// TIA Portal project "MAGNET_ITLK_V15.1" (V15.1)
// Interlocs logic fot the CERN magnet tests

(* hardware
DEVICE "S71500/ET200MP station_1"  S7-1500 station
   slot 0: "Rail_0"  Rack  6ES7 590-1***0-0AA0
   slot 0: "PS 25W 24VDC_1"  PS 25W 24VDC  6ES7 505-0KA00-0AB0  V1.0
   slot 1: "PLC_1"  CPU 1511F-1 PN  6ES7 511-1FK02-0AB0  V2.6
      slot 3: "CPU display_1"  6ES7591-1AA00-0AA0
   slot 2: "DI 32x24VDC HF_1"  DI 32x24VDC HF  6ES7 521-1BL00-0AB0  V2.0
   slot 3: "DQ 32x24VDC/0.5A HF_1"  DQ 32x24VDC/0.5A HF  6ES7 522-1BL01-0AB0  V1.1
   slot 100: "PM 70W 120/230VAC"  PM 70W 120/230VAC  6EP1332-4BA00
*)

// ===== PLC "PLC_1"  CPU 1511F-1 PN =====

VAR_GLOBAL   // PLC tag table "Default tag table"
   "Clock_Byte" AT %MB0 : Byte;
   "Clock_10Hz" AT %M0.0 : Bool;
   "Clock_5Hz" AT %M0.1 : Bool;
   "Clock_2.5Hz" AT %M0.2 : Bool;
   "Clock_2Hz" AT %M0.3 : Bool;
   "Clock_1.25Hz" AT %M0.4 : Bool;
   "Clock_1Hz" AT %M0.5 : Bool;
   "Clock_0.625Hz" AT %M0.6 : Bool;
   "Clock_0.5Hz" AT %M0.7 : Bool;
END_VAR

VAR_GLOBAL CONSTANT   // PLC tag table "ConstDiagnostics"
   "DEV_STATE_OK" : USInt := 1;   // device state ok
   "DEV_STATE_LOST_CON" : USInt := 3;   // device state lost connection
   "DEV_STATE_DISABLED" : USInt := 4;   // device state device disabled
   "DEV_STATE_WAS_FAULT" : USInt := 12;   // device state was fault
   "DEV_STATE_WAS_LOST" : USInt := 13;   // device state connection was lost
   "DEV_STATE_WAS_DISABLED" : USInt := 14;   // device state device was disabled
   "MAX_DEVICES_SYSTEM" : Int := 10;   // max number of devices per IO system
   "MAX_MODULES_DEVICE" : Int := 20;   // max number of modules per device
   "MAX_MODULES_LOCAL" : Int := 15;   // max number of local modules
   "LAST_DEVICE" : Int := -1;   // no next device
   "MAX_SYSTEM" : Int := 2;   // max number of IO system in the project / max number of devices per IO system
   "IO_SYSTEM1" : Int := 1;   // index for IO system 1
   "IO_SYSTEM2" : Int := 2;   // index for IO system 2
   "IO_SYSTEM0" : Int := 0;   // index for local PLC
   "DEV_STATE_FAULT" : USInt := 2;   // device state fault
END_VAR

VAR_GLOBAL   // PLC tag table "ai_dio_tag"
   "DC24V_AUX1_OK" AT %I3.5 : Bool;
   "FLSHBX_HE" AT %Q1.3 : Bool;   // Flashbox Helium
   "KLY_IP_ISn_Current_01" AT %IW304 : Int;
   "KLY_IP_ISn_Current_02" AT %IW306 : Int;
   "KLY_Oil_TSn_SurfTemp" AT %IW222 : Int;
   "KLY_Oil_FSn_WatOutletFlow" AT %IW238 : Int;
   "KLY_Sol_TSn_WatInletTemp" AT %IW216 : Int;
   "KLY_Sol_TSn_WatOutletTemp" AT %IW218 : Int;
   "KLY_Sol_FSn_WatOutletFlow" AT %IW236 : Int;
   "KLY_Sol_TSn_SurfTemp" AT %IW220 : Int;
   "KLY_Win_FSn_WatOutletFlow" AT %IW254 : Int;
   "KLY_Win_TSn_WatOutletTemp" AT %IW214 : Int;
   "KLY_Win_TSn_WatOutletSleeveTemp" AT %IW212 : Int;
   "KLY_Coll_TSn_TopTemp" AT %IW224 : Int;
   "KLY_Coll_TSn_EdgeTemp" AT %IW226 : Int;
   "KLY_Coll_TSn_WatInletTemp" AT %IW248 : Int;
   "KLY_Coll_TSn_WatOutletTemp" AT %IW252 : Int;
   "KLY_Coll_FSn_WatOutletFlow" AT %IW232 : Int;
   "KLY_Body_TSn_WatInletTemp" AT %IW204 : Int;
   "KLY_Body_TSn_WatOutletTemp" AT %IW206 : Int;
   "KLY_Body_FSn_WatOutletFlow" AT %IW234 : Int;
   "KLY_Coll_CollDissipation" AT %IW240 : Int;
   "KLY_Body_BodyDisssipation" AT %IW242 : Int;
   "RFDS_Load_FSn_WatOutletFlow" AT %IW256 : Int;
   "RFDS_Load_TSn_WatOutletTemp" AT %IW250 : Int;
   "spare(7)" AT %Q3.3 : Bool;
   "NO_QUENCH" AT %I3.7 : Bool;   // No quench detected (from safety matrix)
   "DAQ_OK" AT %I1.7 : Bool;   // DAQ system OK
   "PC_1_POWER_FAILURE" AT %I0.6 : Bool;   // Power converter status
   "EE_1_PC_SPA_OK" AT %I0.5 : Bool;   // Slow Power Abort switch OK
   "EE_1_REMOTE" AT %I0.1 : Bool;   // Energy extractionswitches are in remote
   "EE_1_NO_ERROR_CL" AT %I0.2 : Bool;   // Energy extraction switches have nointernalerrors
   "EE_1_CLOSED" AT %I0.3 : Bool;   // Energy extraction keys are closed
   "EE_1_POWER_PERM" AT %I0.0 : Bool;   // Energy extraction switches give power permit
   "KEY2_OK" AT %I1.6 : Bool;   // Cable in parking (0)/ operation (1) position
   "PC_1_CONNECT" AT %I0.7 : Bool;   // Power converter connected (closed contact)
   "PC_1_EXT_OUT" AT %I1.0 : Bool;   // Status of the main circuit breaker of the pwr converter
   "KEY1_OK" AT %I1.5 : Bool;   // Emergency Button OK
   "EE_1_NO_WARNING" AT %I0.4 : Bool;   // Energy Extraction not in warning condition
   "EE_1_FS" AT %I1.1 : Bool;   // EE_1 water flow switch
   "POLSW_1_POS1" AT %I1.2 : Bool;   // Polarity switch 1 position 1
   "EE_2_FS" AT %I3.1 : Bool;   // EE _1water flow switch
   "POLSW_2_POS1" AT %I3.2 : Bool;   // Polarity switch position 1
   "DC24V_AUX2_OK" AT %I3.6 : Bool;   // 24 V PLC power supply ok
   "POLSW_2_POS2" AT %I3.3 : Bool;   // Polarity switch position 2
   "spare(2_4)" AT %I3.4 : Bool;
   "spare3" AT %Q1.0 : Bool;   // Direct power abort
   "PC_1_PERMIT" AT %Q0.3 : Bool;   // Powerconverter permit
   "PC_1_EXT" AT %Q0.4 : Bool;   // Fast Power Abort
   "CLOSE_EE_1" AT %Q0.1 : Bool;   // Close energy extraction switch (action by the operator)
   "EE_1_OPEN_RQ" AT %Q0.0 : Bool;   // Request to open energy extraction switch
   "RESET_EE_1" AT %Q0.2 : Bool;   // Reset energy extraction switch (action by the operator)
   "FLSHBX_HVOLT" AT %Q1.1 : Bool;   // Flashbox High Voltage
   "FLSHBX_HCUR" AT %Q1.2 : Bool;   // Flashbox High Current
   "CPU_Send_RQ" AT %Q3.7 : Bool;
   "MemByteClock7" AT %Q3.6 : Bool;
   "EE_2_OPEN_RQ" AT %Q2.0 : Bool;   // Request to open energy extraction switch
   "CLOSE_EE_2" AT %Q2.1 : Bool;   // Close energy extraction switch (action by the operator)
   "RESET_EE_2" AT %Q2.2 : Bool;   // Reset energy extraction switch (action by the operator)
   "PC_2_PERMIT" AT %Q2.3 : Bool;   // Powerconverter permit
   "PC_2_EXT" AT %Q2.4 : Bool;   // Fast Power Abort
   "EE_2_POWER_PERM" AT %I2.0 : Bool;   // Energy extraction switches give power permit
   "EE_2_REMOTE" AT %I2.1 : Bool;   // Energy extractionswitches are in remote
   "EE_2_NO_ERROR_CL" AT %I2.2 : Bool;   // Energy extraction switches have nointernalerrors
   "EE_2_CLOSED" AT %I2.3 : Bool;   // Energy extraction keys are closed
   "EE_2_NO_WARNING" AT %I2.4 : Bool;   // Energy Extraction not in warning condition
   "EE_2_PC_SPA_OK" AT %I2.5 : Bool;   // Slow Power Abort switch OK
   "PC_2_POWER_FAILURE" AT %I2.6 : Bool;   // Power converter status
   "PC_2_CONNECT" AT %I2.7 : Bool;   // Power converter connected (closed contact)
   "PC_2_EXT_OUT" AT %I3.0 : Bool;   // Status of the main circuit breaker of the pwr converter
   "POLSW_1_POS2" AT %I1.3 : Bool;   // Polarity switch 1 position 2
   "spare(1_4)" AT %I1.4 : Bool;
END_VAR

VAR_GLOBAL CONSTANT   // PLC tag table "ai_dio_tag"
   "DI" : Byte := 1;   // Digital Input type
   "DO" : Byte := 2;   // Digital Output type
   "TSn" : Byte := 1;   // Temperature sensor type
   "PSn" : Byte := 2;   // Pressure sensor type
   "VSn_bipolar_50mV" : Byte := 20;
   "TSn_TC" : Byte := 11;   // Thermocouple - temperature sensor
   "VSn_bipolar_500mV" : Byte := 21;
   "VSn_bipolar_1V" : Byte := 22;
   "VSn_bipolar_5V" : Byte := 23;
   "VSn_bipolar_10V" : Byte := 24;
   "VSn_1_5v" : Byte := 25;
   "VSn_0_10v" : Byte := 3;   // Voltage sensor type
   "ISn_0_20mA" : Byte := 4;
   "ISn_4_20mA" : Byte := 5;
   "FSn_05_80_l_min" : Byte := 6;   // DU06.E.V.R015.A.0 Ultrasonic flowmeter
   "FSn_8_1000_l_min" : Byte := 7;   // DU06.E.V.R050.A.0 Ultrasonic flowmeter
   "PSn_0_10_bar" : Byte := 8;   // PMD02.E.15G.A75.S.I4.K2.0.0 Pressure sensor
   "TSn_0_50_C" : Byte := 9;   // TD20.117 14.111787 - Temperature sensor
   "ISn_bipolar_20mA" : Byte := 26;
   "TSn_PT100" : Byte := 10;   // PT100 - temperature sensor
   "UNKNOW" : Byte := 0;
   "COLL_DISP" : Byte := 12;   // Collector dissipation
   "BODY_DISP" : Byte := 13;   // Body dissipation
   "ISn_IP" : Byte := 27;
   "NORMAL_OPERATION" : Byte := 3;
   "NO_CONVERSION" : Byte := 255;   // Real type - do notdoany conversion
END_VAR

VAR_GLOBAL   // PLC tag table "IOs"
   "FIL_I_REG" AT %M300.0 : Bool;
   "FIL_VMON" AT %MW302 : Int;
   "FIL_IMON" AT %IW314 : Int;
   "FIL_WMON" AT %IW312 : Int;
   "FIL_OUT_LOC_REM" AT %M350.2 : Bool;
   "FIL_OUT_VPGM" AT %MW352 : Int;
   "FIL_START_COMMAND" AT %M300.4 : Bool;
   "FIL_STOP_COMMAND" AT %M300.5 : Bool;
   "SOL1_I_REG" AT %M308.0 : Bool;
   "SOL1_LOC_REM" AT %M308.2 : Bool;
   "SOL1_FAULT" AT %M308.3 : Bool;
   "SOL1_START_COMMAND" AT %M308.4 : Bool;
   "SOL1_STOP_COMMAND" AT %M308.5 : Bool;
   "SOL1_VMON" AT %IW296 : Int;
   "SOL1_IMON" AT %IW300 : Int;
   "SOL1_WMON" AT %MW304 : Int;
   "SOL1_OUT_RESET" AT %M356.1 : Bool;
   "SOL1_OUT_VPGM" AT %MW358 : Int;
   "SOL1_OUT_IPGM" AT %QW6 : Int;
   "FIL_OUT_IPGM" AT %QW4 : Int;
   "SOL2_OUT_IPGM" AT %QW8 : Int;
   "SOL2_VMON" AT %IW298 : Int;
   "SOL2_IMON" AT %IW302 : Int;
   "SOL2_START_COMMAND" AT %M308.6 : Bool;
   "SOL2_STOP_COMMAND" AT %M308.7 : Bool;
END_VAR

VAR_GLOBAL CONSTANT   // PLC tag table "IOs"
   "ENG_0-30A" : Byte := 30;
   "ENG_0-900W" : Byte := 31;
   "PSU_KLYSTRON_SOLENOID" : Int := 2;
   "ENG_0-17A" : Byte := 18;
   "ENG_0-300V" : Byte := 19;
END_VAR

VAR_GLOBAL   // PLC tag table "MachineState"
   "mbi_auxPre" AT %M7.0 : Bool;
   "mbi_filPre" AT %M7.1 : Bool;
   "mbi_stbyPre" AT %M7.3 : Bool;
   "mbi_hvonPre" AT %M7.4 : Bool;
   "mbi_rfonPre" AT %M7.5 : Bool;
   "mw_setState" AT %MW10 : Int;
   "mbi_auxSup" AT %M7.6 : Bool;
   "mbi_filSup" AT %M7.7 : Bool;
   "mbi_stbySup" AT %M8.0 : Bool;
   "mbi_hvonSup" AT %M8.1 : Bool;
   "mbi_rfonSup" AT %M8.2 : Bool;
   "mbi_filPreReady" AT %M7.2 : Bool;
   "mb_location" AT %MB20 : Byte;
   "mb_actState" AT %MB21 : Byte;
   "mbi_aux" AT %M8.4 : Bool;
   "mbi_fil" AT %M8.5 : Bool;
   "mbi_stdby" AT %M8.6 : Bool;
   "mbi_hvon" AT %M8.7 : Bool;
   "mbi_rfon" AT %M9.0 : Bool;
   "t_filHeatingDelay" AT %M9.1 : Bool;
   "t_auxSup" AT %T10 : Timer;
   "t_filSup" AT %T11 : Timer;
   "t_stdbySup" AT %T12 : Timer;
   "t_hvonSup" AT %T13 : Timer;
   "t_rfonSup" AT %T14 : Timer;
END_VAR

TYPE "CommParam"
VERSION : 0.1
   STRUCT
      interface_id : Word;   // HW-identifier of IE-interface submodule
      conn_id : Word;   // Connection reference / identifier
      connection_type : Byte := 16#000B;   // Type of connection: 11=TCP/IP, 19=UDP (17=TCP/IP) ??B#16#11??
      active_established : Bool := False;   // active/passive connection establishment
      local_port : UInt;   // local UDP/TCP port number
      init_com : Bool;   // send_db : INT; recv_db : INT;
      send_len : UDInt;
      recv_len : UDInt;
      sendtrigger : Bool;
      sendtime : Time;
      sendinterval : DInt;
   END_STRUCT;
END_TYPE

TYPE "PSU_Inputs"
VERSION : 0.1
   STRUCT
      I_REG : Bool;   // Signal from PSU, PSU is in constant current mode
      ON_STATUS : Bool;   // Signal from PSU, PSU is truned ON
      LOC_REM : Bool;   // Signal from PSU, TRUE=REMOTE,FALSE=LOCAL
      FAULT : Bool;   // Signal from PSU, TRUE=PSU OK
      VMON : Int;   // Value from PSU, Actual Voltage (V)
      IMON : Int;   // Value from PSU, Actual Current (I)
      WMON : Int;   // Value from PSU, Actual Power (W)
   END_STRUCT;
END_TYPE

TYPE "PSU_Outputs"
VERSION : 0.1
   STRUCT
      ENA_IN : Bool;   // Enable/Disable Power Supply
      RESET : Bool;   // Fault reset
      LOC_REM : Bool;   // LOCAL/REMOTE mode
      VPGM : Int;   // Voltage Setpoint
      IPGM : Int;   // Current Setpoint
   END_STRUCT;
END_TYPE

TYPE "FILAMENT_RST"
VERSION : 0.1
   STRUCT
      ON_STATUS : Bool;   // PSU is Operating normally
      STARTED : Bool;   // PSU has received the ON Command
      STOPPED : Bool;   // PSU is NOT operating
      WARMUP : Bool;   // PSU start procedure is running
      TEMP_REACHED : Bool;   // PSU is at operating temperature - Warmup Done
      I_REG : Bool;   // HIGH= the PSU is in constant cuttent mode
      LOC_REM_ST : Bool;   // HIGH=REMOTE,FALSE=LOCAL
      N_LATCH : Bool;   // Disable Latching from PLC code
      N_FORCE : Bool;   // Disable forcing from PLC code
      IsFIRST : Bool;   // Is the PSU Interlock the first Interlock?
      WARNING : Bool;   // PSU Warning Bit
      INTERLOCK : Bool;   // PSU Interlock Bit
      FORCE_ON : Bool;   // Feedback ForceON
      S_ON_STATUS : Bool;   // Feedback ON_STATUS input
      S_I_REG : Bool;   // Feedback I_REG input
      S_FAULT : Bool;   // Feedback FAULT input
      S_LOC_REM : Bool;   // Feedback LOC_REM input
      I_RAMP_ON : Bool;   // Feedback for Current Ramp ON
      V_RAMP_ON : Bool;   // Feedback for Voltage Ramp ON
      DTYP : Byte;   // PSU Type
      ERR : Word;   // Different error bits stored in the word descibed in the code
      TOTAL_WARMUP_LEFT : Real;   // How much time is left before operation
      WARMUP_LEFT_SP : Real;   // How much time is left before actual SetPoint reached
      UPTIME_NO_HV : Real;   // PSU uptime without HighVoltage
      TIME_COLD_SP1 : Real;   // Feedback Setpoint1 Time
      TIME_COLD_SP2 : Real;   // Feedback Setpoint2 Time
      TIME_COLD_SP3 : Real;   // Feedback Setpoint3 Time
      TIME_WARM_SP1 : Real;   // Feedback Setpoint1 Time warm
      TIME_WARM_SP2 : Real;   // Feedback Setpoint2 Time warm
      TIME_WARM_SP3 : Real;   // Feedback Setpoint3 Time warm
      ACT_SP : Real;   // Actual Setpoint number
      I_RAMP_RATE : Real;   // Feedback Calculated Current Ramp Rate
      V_RAMP_RATE : Real;   // Feedback Calculated Voltage Ramp Rate
      VMON : Real;   // Actual Voltage (V)
      IMON : Real;   // Actual Current (I)
      WMON : Real;   // Actual Power (W)
      S_VMON : Real;   // Feedback VMON input
      S_IMON : Real;   // Feedback IMON input
      S_WMON : Real;   // Feedback WMON input
      I_SP1 : Real;   // Feedback Setpoint1 Current
      I_SP2 : Real;   // Feedback Setpoint2 Current
      I_SP3 : Real;   // Feedback Setpoint3 Current
      V_SP1 : Real;   // Feedback Setpoint1 Voltage
      V_SP2 : Real;   // Feedback Setpoint2 Voltage
      V_SP3 : Real;   // Feedback Setpoint3 Voltage
      I_HIHI : Real;   // Feedback Current Alarm High
      I_LOLO : Real;   // Feedback Current Alarm Low
      I_HIGH : Real;   // Feedback Current Warning High
      I_LOW : Real;   // Feedback Current Warning Low
      W_HIHI : Real;   // Feedback Power Alarm High
      W_LOLO : Real;   // Feedback Power Alarm Low
      W_HIGH : Real;   // Feedback Power Warning High
      W_LOW : Real;   // Feedback Power Warning Low
      I_EGU_SP : Real;   // CurrentSetpoint in engunit
      FIL_MAX_I : Real;   // The maximum allowed Filament current hardwired in the PSU code
      FIL_MAX_W : Real;   // The maximum allowed Filament power hardwired in the PSU code
      TOL_InWARMUP : Real;   // Feedback for Tolareance during Warmup between IMON and IPGM
      TMPST : Date_And_Time;   // Last Interlock or Warning Timestamp
      TOTAL_WARMPUP_T : S5Time;   // Sum of the SetPoints time
   END_STRUCT;
END_TYPE

TYPE "CPU_WCONF"
VERSION : 0.0
   STRUCT
      RESET : Bool;   // CPU reset command
      OFF : Bool;   // OFF Command
      EE_1_CLOSE : Bool;   // Auxiliary Command
      EE_1_RESET : Bool;   // Filament Command
      EE_2_CLOSE : Bool;   // Standby command
      EE_2_RESET : Bool;   // High-voltage ON command
      RFON : Bool;   // RF ON command
      TEST_ALL_AD : Bool;   // Test all arc detectors
      WR_DATA : Bool;   // Write data into the read DB
      OP_MODE : Byte;   // 1 = Bypass mode, 2 = Maintenance/testing mode, 3 = Normal operation, 4 = Wire test
   END_STRUCT;
END_TYPE

TYPE "FILAMENT_WST"
VERSION : 0.1
   STRUCT
      START : Bool;   // Start PSU operation. TRUE=ENABLED
      STOP : Bool := false;   // Stop PSU and reset Timers TRUE = STOP
      FORCE : Bool;   // Force PSU block TRUE = FORCE all inputs
      S_ON_STATUS : Bool;   // Force ON_STATUS input
      S_IVAL : Bool;   // Force I_REG input
      S_LOC_REM : Bool;   // Force LOC_REM input
      S_FAULT : Bool;   // Force FAULT input
      I_RAMP_ON : Bool;   // Enable ramping for Current SP
      V_RAMP_ON : Bool;   // Enable ramping for Voltage SP
      RESET : Bool;   // Reset PSU
      WR_DATA : Bool;   // Write data into the read DB
      TIME_COLD_SP1 : Real;   // Setpoint1 Time
      TIME_COLD_SP2 : Real;   // Setpoint2 Time
      TIME_COLD_SP3 : Real;   // Setpoint3 Time
      TIME_WARM_SP1 : Real;   // Setpoint1 Time if the PSU is already warm
      TIME_WARM_SP2 : Real;   // Setpoint2 Time if the PSU is already warm
      TIME_WARM_SP3 : Real;   // Setpoint3 Time if the PSU is already warm
      I_SP1 : Real;   // Setpoint1 Current
      I_SP2 : Real;   // Setpoint2 Current
      I_SP3 : Real;   // Setpoint3 Current
      V_SP1 : Real;   // Setpoint1 Voltage
      V_SP2 : Real;   // Setpoint2 Voltage
      V_SP3 : Real;   // Setpoint3 Voltage
      S_VMON : Real;   // Force VMON input
      S_IMON : Real;   // Force IMON input
      S_WMON : Real;   // Force WMON input
      V_RAMP_RATE : Real;   // Voltage Ramp rate unit/sec (not used now)
      I_RAMP_RATE : Real;   // Current Ramp rate unit/sec (not used now)
      I_HIHI : Real;   // Current Alarm High
      I_LOLO : Real;   // Current Alarm Low
      I_HIGH : Real;   // Current Warning High
      I_LOW : Real;   // Current Warning Low
      W_HIHI : Real;   // Power Alarm High
      W_LOLO : Real;   // Power Alarm Low
      W_HIGH : Real;   // Power Warning High
      W_LOW : Real;   // Power Warning Low
      TOL_InWARMUP_SP : Real;   // Maximum allowed difference between IMON and IPGM
   END_STRUCT;
END_TYPE

TYPE "CPU_RCONF"
VERSION : 0.0
   STRUCT
      RESET : Bool;   // CPU reset command
      LATCH_MODE : Bool;   // CPU latching mode
      INTERLOCK : Bool;   // CPU Interlock/Alarm
      ACK_REQ : Bool;   // CPU Warning
      GERSEMI_COM_OK : Bool;   // Communication with Gersemi OK
      FLSHBX_HV : Bool;   // Flash Box High Voltage
      FLSHBX_HC : Bool;   // Flash Box High Current
      FLSHBX_He : Bool;   // Flash Box Helium
      RFON_MISS_COND : Bool;   // RF Enable missed condition
      AUX_SUP_COND : Bool;   // AUX missed supervision
      FIL_SUP_COND : Bool;   // FIL missed supervision
      STDBY_SUP_COND : Bool;   // STDBY missed supervision
      HVON_SUP_COND : Bool;   // HVON missed supervision
      RFON_SUP_COND : Bool;   // RFON missed supervision
      OFF : Bool;   // OFF Command
      EE_1_CLOSE : Bool;   // Auxiliary Command
      EE_1_RESET : Bool;   // Filament Command
      EE_2_CLOSE : Bool;   // Standby command
      EE_2_RESET : Bool;   // High-voltage ON command
      RFON : Bool;   // RF ON command
      FORCE_DIS_MODE_ACT : Bool;   // One or more signals are being disabled or forced
      TEST_ALL_AD : Bool;   // Test all arc detectors
      ACT_STAT : Byte;   // Actual State
      SET_STATE : Int;   // Set State to the target
      OP_MODE : Byte;   // 1 = Bypass mode, 2 = Maintenance/testing mode, 3 = Normal operation, 4 = Wire test
   END_STRUCT;
END_TYPE

// folder: Diagnostics

TYPE "typeShowModul"
VERSION : 0.1
   STRUCT
      slotUsed : Bool;   // TRUE if slot is used
      slotErrorState : Bool;   // error state of module
   END_STRUCT;
END_TYPE

TYPE "typeIoSystem"
VERSION : 0.1
   STRUCT
      ioSystemId : UInt;   // ID of IO System
      ioSystemError : Bool;   // TRUE: if an error is occured in the assigned IO System
      firstDevice : Int := 0;   // device number (index) of first device in IO System
      lastDevice : Int := 0;   // device number (index) of last device IO System
      actualConfiguredDevices : Int := 0;   // Actual number of configured devices in the IO System
      device : Array[1.."MAX_DEVICES_SYSTEM"] of "typeDevice";   // List of all devices in the IO System
   END_STRUCT;
END_TYPE

TYPE "typeDevice"
VERSION : 0.1
   STRUCT
      laddr : Hw_Device;   // Logical address of a device or slave (system constant in HW configuration)
      "name" : String[50];   // Device name
      errorState : USInt;   // Status of the device 1=ok!, 2=faulty, 3=lost connection, 4=disabled, 12= was faulty, 13=was lost, 14=was disabled
      error : Bool;   // Signalizes an error in the device/slave
      nextDevice : Int;   // device number of next device
      actualConfiguredModules : Int;   // Actual number of configured modules in the device
      slot : Array[0.."MAX_MODULES_DEVICE"] of "typeModul";   // slot informations
   END_STRUCT;
END_TYPE

TYPE "typeShowDevice"
VERSION : 0.1
   STRUCT
      stationNumber : UInt;   // Station Number of interfaces in HW configuration
      "name" : String[50];   // Device name
      errorState : USInt;   // Status of the device 1=ok!, 2=faulty, 3=lost connection, 4=disabled, 12= was faulty, 13=was lost, 14=was disabled
      slot : Array[0.."MAX_MODULES_DEVICE"] of "typeShowModul";   // slot informations
   END_STRUCT;
END_TYPE

TYPE "typeModul"
VERSION : 0.1
   STRUCT
      slotLaddr : Hw_Io;   // Hardware ID of module
      slotErrorState : Bool;   // error state of module
   END_STRUCT;
END_TYPE

TYPE "typePlc"
VERSION : 0.1
   STRUCT
      actualConfiguredCentralModules : Int;   // Actual number of configured local modules
      errorState : Bool;   // Status of the device 1=ok!, 2=faulty, 3=lost connection, 4=disabled, 12= was faulty, 13=was lost, 14=was disabled
      slot : Array[1.."MAX_MODULES_LOCAL"] of "typeModul";   // slot informations
   END_STRUCT;
END_TYPE

TYPE "typeShowIoSystem"
VERSION : 0.1
   STRUCT
      device : Array[1.."MAX_DEVICES_SYSTEM"] of "typeShowDevice";   // devices informations
   END_STRUCT;
END_TYPE

TYPE "typeShowPlc"
VERSION : 0.1
   STRUCT
      diagnosisLoaded : Bool;   // PLC overview on HMI visible
      errorState : Bool;   // TRUE if the PLC or at least one of the modules is faulty
      slot : Array[1.."MAX_MODULES_LOCAL"] of "typeShowModul";   // module informations
   END_STRUCT;
END_TYPE

TYPE "typeShowActIoSystem"
VERSION : 0.1
   STRUCT
      diagnosisLoaded : Bool;   // IO System overview on HMI visible
      actIoSystem : Int := 1;   // number of selected IO System
      actDeviceIndex : Int;   // number of selected device
      copyModuleStates : Bool;   // is set on HMI to copy module information
      resetStates : Bool;   // is set on HMI to reset saved error states
      device : Array[1.."MAX_DEVICES_SYSTEM"] of "typeShowDevice";   // devices information of selected IO System
      actDevice : "typeShowDevice";   // device information of selected device
   END_STRUCT;
END_TYPE

// folder: PowerSupply

TYPE "SOLENOID_RST"
VERSION : 0.1
   STRUCT
      ON_STATUS : Bool;   // PSU is Operating normally
      STARTED : Bool;   // PSU has received the ON Command
      STOPPED : Bool;   // PSU is NOT operating
      I_REG : Bool;   // HIGH= the PSU is in constant cuttent mode
      LOC_REM_ST : Bool;   // HIGH=REMOTE,FALSE=LOCAL
      N_LATCH : Bool;   // Disable Latching from PLC code
      N_FORCE : Bool;   // Disable forcing from PLC code
      IsFIRST : Bool;   // Is the PSU Interlock the first Interlock?
      WARNING : Bool;   // PSU Warning Bit
      INTERLOCK : Bool;   // PSU Interlock Bit
      FORCE_ON : Bool;   // Feedback ForceON
      S_ON_STATUS : Bool;   // Feedback ON_STATUS input
      S_IREG : Bool;   // Feedback I_REG input
      S_FAULT : Bool;   // Feedback FAULT input
      S_LOC_REM : Bool;   // Feedback LOC_REM input
      DTYP : Byte;   // PSU Type
      ERR : Word;   // Different error bits stored in the word descibed in the code
      UPTIME_NO_HV : DWord;   // PSU uptime without HighVoltage
      VMON : Real;   // Actual Voltage (V)
      IMON : Real;   // Actual Current (I)
      S_VMON : Real;   // Feedback VMON input
      S_IMON : Real;   // Feedback IMON input
      I_SP : Real;   // Feedback Setpoint Current
      V_SP : Real;   // Feedback Setpoint Voltage
      I_HIHI : Real;   // Feedback Current Alarm High
      I_LOLO : Real;   // Feedback Current Alarm Low
      I_HIGH : Real;   // Feedback Current Warning High
      I_LOW : Real;   // Feedback Current Warning Low
      V_HIHI : Real;   // Feedback Voltage Alarm High
      V_LOLO : Real;   // Feedback Voltage Alarm Low
      V_HIGH : Real;   // Feedback Voltage Warning High
      V_LOW : Real;   // Feedback Voltage Warning Low
      V_EGU_SP : Real;   // Voltage Setpoint in engunit
      I_EGU_SP : Real;   // CurrentSetpoint in engunit
      TMPST : Date_And_Time;   // Last Interlock or Warning Timestamp
      SOL_MAX_I : Real;   // The maximum allowed Solenoid current hardwired in the PSU code
      SOL_MAX_V : Real;   // The maximum allowed Solenoid voltage hardwired in the PSU code
   END_STRUCT;
END_TYPE

TYPE "SOLENOID_WST"
VERSION : 0.1
   STRUCT
      START : Bool;   // Start PSU operation. TRUE=ENABLED
      STOP : Bool := false;   // Stop PSU and reset Timers TRUE = STOP
      FORCE : Bool;   // Force PSU block TRUE = FORCE all inputs
      S_ON_STATUS : Bool;   // Force ON_STATUS input
      S_IREG : Bool;   // Force I_REG input
      S_LOC_REM : Bool;   // Force LOC_REM input
      S_FAULT : Bool;   // Force FAULT input
      RESET : Bool;   // Reset PSU
      WR_DATA : Bool;   // Write data into the read DB
      I_SP : Real;   // Setpoint Current
      V_SP : Real;   // Setpoint Voltage
      S_VMON : Real;   // Force VMON input
      S_IMON : Real;   // Force IMON input
      I_HIHI : Real;   // Current Alarm High
      I_LOLO : Real;   // Current Alarm Low
      I_HIGH : Real;   // Current Warning High
      I_LOW : Real;   // Current Warning Low
      V_HIHI : Real;   // Voltage Alarm High
      V_LOLO : Real;   // Voltage Alarm Low
      V_HIGH : Real;   // Voltage Warning High
      V_LOW : Real;   // Voltage Warning Low
   END_STRUCT;
END_TYPE

// folder: SignalProcessing

TYPE "DIO_WST"
VERSION : 0.1
   STRUCT
      DISABLE : Bool;   // Disable the variable
      FORCE : Bool;   // Force the variable to Force_To
      SVAL : Bool;   // Simlation Value
      WR_DATA : Bool;   // Write data into the read DB
   END_STRUCT;
END_TYPE

TYPE "DATE"
VERSION : 0.1
   STRUCT
      "Time" : Date_And_Time;
   END_STRUCT;
END_TYPE

TYPE "DIO_RST"
VERSION : 0.1
   STRUCT
      VAL : Bool;   // Field value
      INTERLOCK : Bool;   // Alarm/Interlock variable
      SVAL : Bool;   // Simulation Value
      DISABLE : Bool;   // Disable the variable
      FORCE : Bool;   // Force the variable to Force_To
      N_FORCE : Bool;   // Cannot force
      N_LATCH : Bool;   // Never latch
      IsFIRST : Bool;   // First variable interlocked before the CPU alarm trips
      INVERT : Bool;   // Invert Digital Output Field Value
      TMPST : Date_And_Time;   // Time-stamp
      DTYP : Byte;   // Device type
      ERR : Byte;   // Error code
   END_STRUCT;
END_TYPE

TYPE "AF_WST"
VERSION : 0.0
   STRUCT
      DISABLE : Bool;   // Variable disable
      FORCE : Bool;   // Force the variable to the simulation value
      WR_DATA : Bool;   // Write data into the read DB
      HIHI : Real;   // Hihi Alarm limit
      HIGH : Real;   // High Alarm limit
      LOW : Real;   // Low Alarm limit
      LOLO : Real;   // Lolo Alarm limit
      AOFF : Real;   // Adjustment Offset
      SVAL : Real;   // Simulation Value
   END_STRUCT;
END_TYPE

TYPE "AF_RST"
VERSION : 0.0
   STRUCT
      WARNING : Bool;   // Warning flag
      INTERLOCK : Bool;   // Alarm/Interlock
      DISABLE : Bool;   // Variable disable
      FORCE : Bool;   // Force the variable to the simulation value
      N_FORCE : Bool;   // Cannot force
      N_LATCH : Bool;   // Never Latch
      IsFIRST : Bool;   // First variable interlocked before the CPU alarm trips
      LOW_ALARM : Bool;   // Low alarm detection
      HIGH_ALARM : Bool;   // High alarm detection
      TMPST : Date_And_Time;   // Time-stamp
      DTYP : Byte;   // Device type
      ERR : Word;   // Error code
      HIHI : Real;   // Hihi Alarm limit
      HIGH : Real;   // High Alarm limit
      LOW : Real;   // Low Alarm limit
      LOLO : Real;   // Lolo Alarm limit
      AOFF : Real;   // Adjustment Offset
      SVAL : Real;   // Simulation Value
      EGU : Real;   // Engineering Field Unit
      VAL : Int;   // Field Value
   END_STRUCT;
END_TYPE

// folder: Diagnostics

DATA_BLOCK "PlcStatus"   // DB1
{ S7_Optimized_Access := 'TRUE' }
VERSION : 0.1
   VAR
      plc : "typePlc";
   END_VAR
BEGIN
END_DATA_BLOCK

DATA_BLOCK "InstDiagnostics"   // DB2000
{ S7_Optimized_Access := 'TRUE' }
VERSION : 0.1
// stored: InstanceOfName Diagnostics
"Diagnostics"
BEGIN
END_DATA_BLOCK

DATA_BLOCK "InstDiagStartupIoSystem"   // DB2001
{ S7_Optimized_Access := 'TRUE' }
VERSION : 0.1
// stored: InstanceOfName DiagStartupIoSystem
"DiagStartupIoSystem"
BEGIN
END_DATA_BLOCK

DATA_BLOCK "InstDiagStartupPlc"   // DB2002
{ S7_Optimized_Access := 'TRUE' }
VERSION : 0.1
// stored: InstanceOfName DiagStartupPlc
"DiagStartupPlc"
BEGIN
END_DATA_BLOCK

DATA_BLOCK "DiagnosticsData"   // DB2080
TITLE = Diagosis data DB
{ S7_Optimized_Access := 'TRUE' }
AUTHOR : SIEMENS
FAMILY : Diagnose
NAME : 10
VERSION : 0.1
// The global data block contains the data structure of the IO system, the control, the devices with the modules and an error buffer.
   VAR
      plc : "typePlc";   // diagnosis information PLC
      ioSystem : Array[1.."MAX_SYSTEM"] of "typeIoSystem";   // diagnosis information IO systems
   END_VAR
BEGIN
END_DATA_BLOCK

DATA_BLOCK "HmiDB"   // DB2081
{ S7_Optimized_Access := 'TRUE' }
VERSION : 0.1
   VAR
      showPlc : "typeShowPlc";   // diagnosis information PLC for visualisation
      showIoSystem : Array[1.."MAX_SYSTEM"] of "typeShowIoSystem";   // diagnosis information IO systems for visualisation
      showActIoSystem : "typeShowActIoSystem";   // diagnosis information selected IO systems for visualisation
   END_VAR
BEGIN
END_DATA_BLOCK

// folder: EPICS_Communication

DATA_BLOCK "CH_PARAM_TCP_CPU"   // DB300
{ S7_Optimized_Access := 'FALSE' }
VERSION : 0.1
   VAR
      CommParam : "CommParam";
   END_VAR
BEGIN
   CommParam.send_len := 8;
   CommParam.recv_len := 4;
   CommParam.sendinterval := DINT#500;
   CommParam.local_port := 3000;
   CommParam.interface_id := 64;
   CommParam.conn_id := 3;
END_DATA_BLOCK

DATA_BLOCK "CH_PARAM_TCP_AF"   // DB301
{ S7_Optimized_Access := 'FALSE' }
VERSION : 0.1
   VAR
      CommParam : "CommParam";
   END_VAR
BEGIN
   CommParam.send_len := 1232;
   CommParam.recv_len := 728;
   CommParam.sendinterval := DINT#500;
   CommParam.local_port := 3001;
   CommParam.interface_id := 64;
   CommParam.conn_id := 4;
END_DATA_BLOCK

DATA_BLOCK "CH_PARAM_TCP_DIO"   // DB302
{ S7_Optimized_Access := 'FALSE' }
VERSION : 0.1
   VAR
      CommParam : "CommParam";
   END_VAR
BEGIN
   CommParam.send_len := 912;
   CommParam.recv_len := 152;
   CommParam.sendinterval := DINT#500;
   CommParam.local_port := 3002;
   CommParam.interface_id := 64;
   CommParam.conn_id := 5;
END_DATA_BLOCK

DATA_BLOCK "CH_PARAM_TCP_PSU"   // DB303
{ S7_Optimized_Access := 'FALSE' }
VERSION : 0.1
   VAR
      CommParam : "CommParam";
   END_VAR
BEGIN
   CommParam.send_len := 430;
   CommParam.recv_len := 256;
   CommParam.sendinterval := DINT#500;
   CommParam.local_port := 3003;
   CommParam.interface_id := 64;
   CommParam.conn_id := 6;
END_DATA_BLOCK

DATA_BLOCK "TCP1_instance"   // DB310
{ S7_Optimized_Access := 'FALSE' }
AUTHOR : CSL
FAMILY : TSTMP
NAME : S_R_TCP1
VERSION : 1.0
// stored: InstanceOfName Tsend_Trecv
"Tsend_Trecv"
BEGIN
END_DATA_BLOCK

DATA_BLOCK "TCP2_instance"   // DB311
{ S7_Optimized_Access := 'FALSE' }
AUTHOR : CSL
FAMILY : TSTMP
NAME : S_R_TCP1
VERSION : 1.0
// stored: InstanceOfName Tsend_Trecv
"Tsend_Trecv"
BEGIN
END_DATA_BLOCK

DATA_BLOCK "TCP3_instance"   // DB312
{ S7_Optimized_Access := 'FALSE' }
AUTHOR : CSL
FAMILY : TSTMP
NAME : S_R_TCP1
VERSION : 1.0
// stored: InstanceOfName Tsend_Trecv
"Tsend_Trecv"
BEGIN
END_DATA_BLOCK

DATA_BLOCK "TCP4_instance"   // DB313
{ S7_Optimized_Access := 'FALSE' }
AUTHOR : CSL
FAMILY : TSTMP
NAME : S_R_TCP1
VERSION : 1.0
// stored: InstanceOfName Tsend_Trecv
"Tsend_Trecv"
BEGIN
END_DATA_BLOCK

// folder: Gersemi_Communication

DATA_BLOCK "Data_from_Gersemi"   // DB401
{ S7_Optimized_Access := 'FALSE' }
VERSION : 0.1
   VAR
      NDR : Bool;   // Data ready
      ERR : Bool;   // Error
      Gersemi_CommOK : Bool;
      mem1_6sec : Bool;
      memDoneStat : Word;   // Status word
      memErrStat : Word;
      LastHeartBeat : Int;   // Heart Beat From Gersemi
      HeartBeat : Int;   // HeartBeat to compare with
      "Cryo_1,9K" : Bool;
      "Cryo_4,5K" : Bool;
      Cryo_leads_OK : Bool;
      Lead_1_T_OK : Bool;
      Lead_2_T_OK : Bool;
      Lead_3_T_OK : Bool;
      Lead_4_T_OK : Bool;
      Lead_1_V_OK : Bool;
      Lead_2_V_OK : Bool;
      Lead_3_V_OK : Bool;
      Lead_4_V_OK : Bool;
      spareBit_4 : Bool;
      spareBit_5 : Bool;
      spareBit_6 : Bool;
      spareBit_7 : Bool;
      spareBit_8 : Bool;
      r1 : Real;   // Data
      r2 : Real;
      r3 : Real;
      r4 : Real;
      r5 : Real;
      r6 : Real;
      r7 : Real;
      r8 : Real;
   END_VAR
BEGIN
END_DATA_BLOCK

// folder: PowerSupply

DATA_BLOCK "PSU_RDATA"   // DB3010
{ S7_Optimized_Access := 'FALSE' }
VERSION : 0.1
   VAR
      FILAMENT : "FILAMENT_RST";
      SOLENOID1 : "SOLENOID_RST";
      SOLENOID2 : "SOLENOID_RST";
      SOLENOID3 : "SOLENOID_RST";
   END_VAR
BEGIN
END_DATA_BLOCK

DATA_BLOCK "PSU_WDATA"   // DB3011
{ S7_Optimized_Access := 'FALSE' }
VERSION : 0.1
   VAR
      FILAMENT : "FILAMENT_WST";
      SOLENOID1 : "SOLENOID_WST";
      SOLENOID2 : "SOLENOID_WST";
      SOLENOID3 : "SOLENOID_WST";
   END_VAR
BEGIN
   FILAMENT.V_RAMP_ON := false;
   FILAMENT.TIME_COLD_SP1 := 0.0;
   FILAMENT.TIME_COLD_SP2 := 0.0;
   FILAMENT.TIME_COLD_SP3 := 0.0;
   FILAMENT.TIME_WARM_SP1 := 0.0;
   FILAMENT.TIME_WARM_SP2 := 0.0;
   FILAMENT.TIME_WARM_SP3 := 0.0;
   FILAMENT.I_SP1 := 0.0;
   FILAMENT.I_SP2 := 0.0;
   FILAMENT.I_SP3 := 0.0;
   FILAMENT.TOL_InWARMUP_SP := 5.0;
END_DATA_BLOCK

// folder: SignalProcessing

DATA_BLOCK "DateTime"   // DB50
{ S7_Optimized_Access := 'FALSE' }
VERSION : 0.1
   VAR
      Out_Date : Word;
      Out_Clock_Date : Date_And_Time;
      Out_day_Week : Int;
      Out_Time : Time_Of_Day;
      Out_Clock_Date_Local : Date_And_Time;
   END_VAR
BEGIN
END_DATA_BLOCK

DATA_BLOCK "CPU_RDATA"   // DB200
{ S7_Optimized_Access := 'FALSE' }
VERSION : 0.1
   VAR
      CPU_CONF : "CPU_RCONF";
   END_VAR
BEGIN
   CPU_CONF.LATCH_MODE := true;
END_DATA_BLOCK

DATA_BLOCK "CPU_WDATA"   // DB201
{ S7_Optimized_Access := 'FALSE' }
VERSION : 0.1
   VAR
      CPU_CONF : "CPU_WCONF";
   END_VAR
BEGIN
END_DATA_BLOCK

DATA_BLOCK "AF_RDATA"   // DB202
TITLE = Analog float read data
{ S7_Optimized_Access := 'FALSE' }
VERSION : 0.2
   VAR
      KLY_IP_ISn_Current : "AF_RST";
      KLY_Oil_TSn_SurfTemp : "AF_RST";
      KLY_Oil_FSn_WatOutletFlow : "AF_RST";
      KLY_Oil_TSn_WatInletTemp : "AF_RST";
      KLY_Sol_TSn_WatInletTemp : "AF_RST";
      KLY_Sol_TSn_WatInletTempMan : "AF_RST";
      KLY_Sol_TSn_WatOutletTemp : "AF_RST";
      KLY_Sol_FSn_WatOutletFlow : "AF_RST";
      KLY_Sol_TSn_SurfTemp : "AF_RST";
      KLY_Win_FSn_WatOutletFlow : "AF_RST";
      KLY_Win_TSn_WatOutletTemp : "AF_RST";
      KLY_Win_TSn_WatOutletTempMan : "AF_RST";
      KLY_Win_TSn_WatOutletSleeveTemp : "AF_RST";
      KLY_Coll_TSn_TopTemp : "AF_RST";
      KLY_Coll_TSn_EdgeTemp : "AF_RST";
      KLY_Coll_TSn_WatInletTemp : "AF_RST";
      KLY_Coll_TSn_WatOutletTemp : "AF_RST";
      KLY_Coll_FSn_WatOutletFlow : "AF_RST";
      KLY_Body_TSn_WatInletTemp : "AF_RST";
      KLY_Body_TSn_WatOutletTemp : "AF_RST";
      KLY_Body_FSn_WatOutletFlow : "AF_RST";
      KLY_Coll_CollDissipation : "AF_RST";
      KLY_Body_BodyDisssipation : "AF_RST";
      RFDS_Circ_FSn_WatOutletFlow : "AF_RST";
      RFDS_Circ_TSn_WatInletTemp : "AF_RST";
      RFDS_Load_TSn_WatInletTemp : "AF_RST";
      RFDS_Load_FSn_WatOutletFlow : "AF_RST";
      RFDS_Load_TSn_WatOutletTemp : "AF_RST";
   END_VAR
BEGIN
END_DATA_BLOCK

DATA_BLOCK "AF_WDATA"   // DB203
TITLE = Analog float write data
{ S7_Optimized_Access := 'FALSE' }
VERSION : 0.1
   VAR
      KLY_IP_ISn_Current : "AF_WST";
      KLY_Oil_TSn_SurfTemp : "AF_WST";
      KLY_Oil_FSn_WatOutletFlow : "AF_WST";
      KLY_Oil_TSn_WatInletTemp : "AF_WST";
      KLY_Sol_TSn_WatInletTemp : "AF_WST";
      KLY_Sol_TSn_WatInletTempMan : "AF_WST";
      KLY_Sol_TSn_WatOutletTemp : "AF_WST";
      KLY_Sol_FSn_WatOutletFlow : "AF_WST";
      KLY_Sol_TSn_SurfTemp : "AF_WST";
      KLY_Win_FSn_WatOutletFlow : "AF_WST";
      KLY_Win_TSn_WatOutletTemp : "AF_WST";
      KLY_Win_TSn_WatOutletTempMan : "AF_WST";
      KLY_Win_TSn_WatOutletSleeveTemp : "AF_WST";
      KLY_Coll_TSn_TopTemp : "AF_WST";
      KLY_Coll_TSn_EdgeTemp : "AF_WST";
      KLY_Coll_TSn_WatInletTemp : "AF_WST";
      KLY_Coll_TSn_WatOutletTemp : "AF_WST";
      KLY_Coll_FSn_WatOutletFlow : "AF_WST";
      KLY_Body_TSn_WatInletTemp : "AF_WST";
      KLY_Body_TSn_WatOutletTemp : "AF_WST";
      KLY_Body_FSn_WatOutletFlow : "AF_WST";
      KLY_Coll_CollDissipation : "AF_WST";
      KLY_Body_BodyDisssipation : "AF_WST";
      RFDS_Circ_FSn_WatOutletFlow : "AF_WST";
      RFDS_Circ_TSn_WatInletTemp : "AF_WST";
      RFDS_Load_TSn_WatInletTemp : "AF_WST";
      RFDS_Load_FSn_WatOutletFlow : "AF_WST";
      RFDS_Load_TSn_WatOutletTemp : "AF_WST";
   END_VAR
BEGIN
END_DATA_BLOCK

DATA_BLOCK "DIO_RDATA"   // DB204
TITLE = Digital I/O write data
{ S7_Optimized_Access := 'FALSE' }
VERSION : 0.1
   VAR
      EE_1_POWER_PERM : "DIO_RST";
      EE_1_REMOTE : "DIO_RST";
      EE_1_NO_ERROR_CL : "DIO_RST";
      EE_1_CLOSED : "DIO_RST";
      spare_1 : "DIO_RST";
      EE_1_PC_SPA_OK : "DIO_RST";
      PC_1_POWER_Failure : "DIO_RST";
      PC_1_CONNECT : "DIO_RST";
      PC_1_EXT_OUT : "DIO_RST";
      EE_1_FS : "DIO_RST";
      POLSW_1_POS1 : "DIO_RST";
      POLSW_1_POS2 : "DIO_RST";
      spare_4 : "DIO_RST";
      KEY1_OK : "DIO_RST";
      NO_QUENCH : "DIO_RST";
      DAQ_OK : "DIO_RST";
      EE_2_POWER_PERM : "DIO_RST";
      EE_2_REMOTE : "DIO_RST";
      EE_2_NO_ERROR_CL : "DIO_RST";
      EE_2_CLOSED : "DIO_RST";
      spare_2 : "DIO_RST";
      EE_2_PC_SPA_OK : "DIO_RST";
      PC_2_POWER_Failure : "DIO_RST";
      PC_2_CONNECT : "DIO_RST";
      PC_2_EXT_OUT : "DIO_RST";
      EE_2_FS : "DIO_RST";
      POLSW_2_POS1 : "DIO_RST";
      POLSW_2_POS2 : "DIO_RST";
      spare_8 : "DIO_RST";
      DC24V_AUX1_OK : "DIO_RST";
      DC24V_AUX2_OK : "DIO_RST";
      KEY2_OK : "DIO_RST";
      EE_1_OPEN_RQ : "DIO_RST";
      spare27 : "DIO_RST";
      spare28 : "DIO_RST";
      PC_1_PERMIT : "DIO_RST";
      PC_1_EXT : "DIO_RST";
      spare_9 : "DIO_RST";
      spare_10 : "DIO_RST";
      spare_11 : "DIO_RST";
      spare_3 : "DIO_RST";
      spare31 : "DIO_RST";
      spare32 : "DIO_RST";
      spare33 : "DIO_RST";
      spare_12 : "DIO_RST";
      spare_13 : "DIO_RST";
      spare_14 : "DIO_RST";
      spare_15 : "DIO_RST";
      EE_2_OPEN_RQ : "DIO_RST";
      spare29 : "DIO_RST";
      spare30 : "DIO_RST";
      PC_2_PERMIT : "DIO_RST";
      PC_2_EXT : "DIO_RST";
      spare_16 : "DIO_RST";
      spare_17 : "DIO_RST";
      spare_18 : "DIO_RST";
      spare_19 : "DIO_RST";
      spare_20 : "DIO_RST";
      spare_21 : "DIO_RST";
      spare_22 : "DIO_RST";
      spare_23 : "DIO_RST";
      spare_24 : "DIO_RST";
      spare_25 : "DIO_RST";
      CRYO_LEADS_OK : "DIO_RST";
      LEAD_1_TEMP_OK : "DIO_RST";
      LEAD_2_TEMP_OK : "DIO_RST";
      LEAD_3_TEMP_OK : "DIO_RST";
      LEAD_4_TEMP_OK : "DIO_RST";
      "CRYO_1.9K" : "DIO_RST";
      "CRYO_4.5K" : "DIO_RST";
      CRYO_300K_HE : "DIO_RST";
      CRYO_300K_AIR : "DIO_RST";
      LEAD_1_VOLT_OK : "DIO_RST";
      LEAD_2_VOLT_OK : "DIO_RST";
      LEAD_3_VOLT_OK : "DIO_RST";
      LEAD_4_VOLT_OK : "DIO_RST";
   END_VAR
BEGIN
END_DATA_BLOCK

DATA_BLOCK "DIO_WDATA"   // DB205
TITLE = Digital I/O write data
{ S7_Optimized_Access := 'FALSE' }
VERSION : 0.1
   VAR
      EE_1_POWER_PERM : "DIO_WST";
      EE_1_REMOTE : "DIO_WST";
      EE_1_NO_ERROR_CL : "DIO_WST";
      EE_1_CLOSED : "DIO_WST";
      spare_1 : "DIO_WST";
      EE_1_PC_SPA_OK : "DIO_WST";
      PC_1_POWER_Failure : "DIO_WST";
      PC_1_CONNECT : "DIO_WST";
      PC_1_EXT_OUT : "DIO_WST";
      EE_1_FS : "DIO_WST";
      POLSW_1_POS1 : "DIO_WST";
      POLSW_1_POS2 : "DIO_WST";
      spare_4 : "DIO_WST";
      KEY1_OK : "DIO_WST";
      NO_QUENCH : "DIO_WST";
      DAQ_OK : "DIO_WST";
      EE_2_POWER_PERM : "DIO_WST";
      EE_2_REMOTE : "DIO_WST";
      EE_2_NO_ERROR_CL : "DIO_WST";
      EE_2_CLOSED : "DIO_WST";
      spare_2 : "DIO_WST";
      EE_2_PC_SPA_OK : "DIO_WST";
      PC_2_POWER_Failure : "DIO_WST";
      PC_2_CONNECT : "DIO_WST";
      PC_2_EXT_OUT : "DIO_WST";
      EE_2_FS : "DIO_WST";
      POLSW_2_POS1 : "DIO_WST";
      POLSW_2_POS2 : "DIO_WST";
      spare_8 : "DIO_WST";
      DC24V_AUX1_OK : "DIO_WST";
      DC24V_AUX2_OK : "DIO_WST";
      KEY2_OK : "DIO_WST";
      EE_1_OPEN_RQ : "DIO_WST";
      spare27 : "DIO_WST";
      spare28 : "DIO_WST";
      PC_1_PERMIT : "DIO_WST";
      PC_1_EXT : "DIO_WST";
      spare_9 : "DIO_WST";
      spare_10 : "DIO_WST";
      spare_11 : "DIO_WST";
      spare_3 : "DIO_WST";
      spare31 : "DIO_WST";
      spare32 : "DIO_WST";
      spare33 : "DIO_WST";
      spare_12 : "DIO_WST";
      spare_13 : "DIO_WST";
      spare_14 : "DIO_WST";
      spare_15 : "DIO_WST";
      EE_2_OPEN_RQ : "DIO_WST";
      spare29 : "DIO_WST";
      spare30 : "DIO_WST";
      PC_2_PERMIT : "DIO_WST";
      PC_2_EXT : "DIO_WST";
      spare_16 : "DIO_WST";
      spare_17 : "DIO_WST";
      spare_18 : "DIO_WST";
      spare_19 : "DIO_WST";
      spare_20 : "DIO_WST";
      spare_21 : "DIO_WST";
      spare_22 : "DIO_WST";
      spare_23 : "DIO_WST";
      spare_24 : "DIO_WST";
      spare_25 : "DIO_WST";
      CRYO_LEADS_OK : "DIO_WST";
      LEAD_1_TEMP_OK : "DIO_WST";
      LEAD_2_TEMP_OK : "DIO_WST";
      LEAD_3_TEMP_OK : "DIO_WST";
      LEAD_4_TEMP_OK : "DIO_WST";
      "CRYO_1.9K" : "DIO_WST";
      "CRYO_4.5K" : "DIO_WST";
      CRYO_300K_HE : "DIO_WST";
      CRYO_300K_AIR : "DIO_WST";
      LEAD_1_VOLT_OK : "DIO_WST";
      LEAD_2_VOLT_OK : "DIO_WST";
      LEAD_3_VOLT_OK : "DIO_WST";
      LEAD_4_VOLT_OK : "DIO_WST";
   END_VAR
BEGIN
END_DATA_BLOCK

// folder: System blocks/Program resources

DATA_BLOCK "IEC_Timer_EE1_DB"   // DB2
{ S7_Optimized_Access := 'TRUE' }
AUTHOR : Simatic
FAMILY : IEC
NAME : IEC_TMR
VERSION : 1.0
// stored: InstanceOfName IEC_TIMER
"IEC_TIMER"
BEGIN
END_DATA_BLOCK

DATA_BLOCK "IEC_Timer_EE2_DB"   // DB3
{ S7_Optimized_Access := 'TRUE' }
AUTHOR : Simatic
FAMILY : IEC
NAME : IEC_TMR
VERSION : 1.0
// stored: InstanceOfName IEC_TIMER
"IEC_TIMER"
BEGIN
END_DATA_BLOCK

DATA_BLOCK "T_TestAllAD_DB"   // DB220
{ S7_Optimized_Access := 'TRUE' }
AUTHOR : Simatic
FAMILY : IEC
NAME : IEC_TMR
VERSION : 1.0
// stored: InstanceOfName IEC_TIMER
"IEC_TIMER"
BEGIN
END_DATA_BLOCK

DATA_BLOCK "T_ResetAllAD_DB"   // DB221
{ S7_Optimized_Access := 'TRUE' }
AUTHOR : Simatic
FAMILY : IEC
NAME : IEC_TMR
VERSION : 1.0
// stored: InstanceOfName IEC_TIMER
"IEC_TIMER"
BEGIN
END_DATA_BLOCK

// folder: (top level)

FUNCTION "GET_MEASUREMENT" : Void   // FC12, SCL
{ S7_Optimized_Access := 'FALSE' }
VERSION : 0.1
   VAR_TEMP
      POLSW_INTERLOCK_1 : Bool;   // Polarity switches ok (one open one closed)
      POLSW_INTERLOCK_2 : Bool;
      EE_1_Open_RQ : Bool;
      EE_2_Open_RQ : Bool;
      t1 : Time;
      t2 : Time;
   END_VAR
   VAR CONSTANT
      pulse_time : Time := T#500ms;
   END_VAR
BEGIN
   //Analog signal type

   ////"AF_RDATA".Main_110_PT.DTYP := "TSn_PT100";
   "AF_RDATA".KLY_IP_ISn_Current.DTYP := "ISn_IP";

   "AF_RDATA".KLY_Oil_TSn_SurfTemp.DTYP := "NO_CONVERSION"; // no scaling

   ////"AF_RDATA".Main_110_PT.VAL := "Main_110_PT";
   //
   // Fake data fora test to be deleted !!!!!!!!!!!!!!!!!!!!!!!!!!!!!
   "AF_RDATA".KLY_IP_ISn_Current.VAL := 10;
   "AF_RDATA".KLY_Oil_TSn_SurfTemp.EGU := 1.234; // no scaling

   // "DO_0":P  := "Clock_2Hz";
   // "DO_1":P  := "CH_PARAM_TCP_CPU".CommParam.sendtrigger;
   // "DO_2":P  := "CH_PARAM_TCP_AF".CommParam.sendtrigger;
   // "DO_3":P  := "CH_PARAM_TCP_DIO".CommParam.sendtrigger;

   //Digital Inputs/Outputs type
   //

   "DIO_RDATA"."EE_1_POWER_PERM".VAL := "EE_1_POWER_PERM";
   "DIO_RDATA".EE_1_REMOTE.VAL := "EE_1_REMOTE";
   "DIO_RDATA".EE_1_NO_ERROR_CL.VAL := "EE_1_NO_ERROR_CL";
   "DIO_RDATA"."EE_1_CLOSED".VAL := "EE_1_CLOSED";
   "DIO_RDATA"."spare_1".VAL := "EE_1_NO_WARNING";
   "DIO_RDATA".EE_1_PC_SPA_OK.VAL := "EE_1_PC_SPA_OK";
   "DIO_RDATA".PC_1_POWER_Failure.VAL := "PC_1_POWER_FAILURE";
   "DIO_RDATA".PC_1_CONNECT.VAL := "PC_1_CONNECT";
   "DIO_RDATA".PC_1_EXT_OUT.VAL := "PC_1_EXT_OUT";
   "DIO_RDATA".EE_1_FS.VAL := "EE_1_FS";
   "DIO_RDATA".POLSW_1_POS1.VAL := "POLSW_1_POS1";
   "DIO_RDATA".POLSW_1_POS1.VAL := "POLSW_1_POS2";

   "DIO_RDATA".KEY1_OK.VAL := "KEY1_OK";
   "DIO_RDATA".NO_QUENCH.VAL := "NO_QUENCH";
   "DIO_RDATA".DAQ_OK.VAL := "DAQ_OK";

   "DIO_RDATA"."EE_2_POWER_PERM".VAL := "EE_2_POWER_PERM";
   "DIO_RDATA".EE_2_REMOTE.VAL := "EE_2_REMOTE";
   "DIO_RDATA".EE_2_NO_ERROR_CL.VAL := "EE_2_NO_ERROR_CL";
   "DIO_RDATA"."EE_2_CLOSED".VAL := "EE_2_CLOSED";
   "DIO_RDATA"."spare_2".VAL := "EE_2_NO_WARNING";
   "DIO_RDATA".EE_2_PC_SPA_OK.VAL := "EE_2_PC_SPA_OK";
   "DIO_RDATA".PC_2_POWER_Failure.VAL := "PC_2_POWER_FAILURE";
   "DIO_RDATA".PC_2_CONNECT.VAL := "PC_2_CONNECT";
   "DIO_RDATA".PC_2_EXT_OUT.VAL := "PC_2_EXT_OUT";
   "DIO_RDATA".EE_2_FS.VAL := "EE_2_FS";
   "DIO_RDATA".POLSW_2_POS1.VAL := "POLSW_2_POS1";
   "DIO_RDATA".POLSW_2_POS1.VAL := "POLSW_2_POS2";

   "DIO_RDATA".DC24V_AUX1_OK.VAL := "DC24V_AUX1_OK";
   "DIO_RDATA".DC24V_AUX2_OK.VAL := "DC24V_AUX2_OK";
   "DIO_RDATA".KEY2_OK.VAL := "KEY2_OK";

   // Data read from Gersemi PLC using S7 communication
   // 
   "DIO_RDATA".LEAD_1_TEMP_OK.VAL := "Data_from_Gersemi".Lead_1_T_OK AND "Data_from_Gersemi".Gersemi_CommOK;
   "DIO_RDATA".LEAD_2_TEMP_OK.VAL := "Data_from_Gersemi".Lead_2_T_OK AND "Data_from_Gersemi".Gersemi_CommOK;   
   "DIO_RDATA".LEAD_3_TEMP_OK.VAL := "Data_from_Gersemi".Lead_3_T_OK AND "Data_from_Gersemi".Gersemi_CommOK; 
   "DIO_RDATA".LEAD_4_TEMP_OK.VAL := "Data_from_Gersemi".Lead_4_T_OK AND "Data_from_Gersemi".Gersemi_CommOK;

   "DIO_RDATA"."CRYO_1.9K".VAL := "Data_from_Gersemi"."Cryo_1,9K" AND "Data_from_Gersemi".Gersemi_CommOK;
   "DIO_RDATA"."CRYO_4.5K".VAL := "Data_from_Gersemi"."Cryo_4,5K" AND "Data_from_Gersemi".Gersemi_CommOK;

   "DIO_RDATA".LEAD_1_VOLT_OK.VAL := "Data_from_Gersemi".Lead_1_V_OK AND "Data_from_Gersemi".Gersemi_CommOK;
   "DIO_RDATA".LEAD_2_VOLT_OK.VAL := "Data_from_Gersemi".Lead_2_V_OK AND "Data_from_Gersemi".Gersemi_CommOK;
   "DIO_RDATA".LEAD_3_VOLT_OK.VAL := "Data_from_Gersemi".Lead_3_V_OK AND "Data_from_Gersemi".Gersemi_CommOK;
   "DIO_RDATA".LEAD_4_VOLT_OK.VAL := "Data_from_Gersemi".Lead_4_V_OK AND "Data_from_Gersemi".Gersemi_CommOK;

   "DIO_RDATA".CRYO_300K_HE.VAL := FALSE;          // TODO 
   "DIO_RDATA".CRYO_300K_AIR.VAL := FALSE;         // TODO 

   "DIO_RDATA".CRYO_LEADS_OK.VAL := "Data_from_Gersemi".Cryo_leads_OK AND "Data_from_Gersemi".Gersemi_CommOK;  

   "CPU_RDATA".CPU_CONF.GERSEMI_COM_OK := "Data_from_Gersemi".Gersemi_CommOK;

   // Type definition: DI/DO required, optional: INVERT (all default false)
   // 
   // Hardware DI
   "DIO_RDATA".EE_1_POWER_PERM.DTYP := "DI";
   "DIO_RDATA".EE_1_POWER_PERM.INVERT := TRUE;
   "DIO_RDATA".EE_1_REMOTE.DTYP := "DI";
   "DIO_RDATA".EE_1_REMOTE.INVERT := TRUE;
   "DIO_RDATA"."EE_1_NO_ERROR_CL".DTYP := "DI";
   "DIO_RDATA"."EE_1_NO_ERROR_CL".INVERT := TRUE;
   "DIO_RDATA".EE_1_CLOSED.DTYP := "DI";
   "DIO_RDATA".EE_1_CLOSED.INVERT := TRUE;
   "DIO_RDATA"."spare_1".DTYP := "DI";
   "DIO_RDATA"."spare_1".INVERT := TRUE;
   "DIO_RDATA".EE_1_PC_SPA_OK.DTYP := "DI";
   "DIO_RDATA".EE_1_PC_SPA_OK.INVERT := TRUE;
   "DIO_RDATA".PC_1_POWER_Failure.DTYP := "DI";
   "DIO_RDATA".PC_1_POWER_Failure.INVERT := TRUE;
   "DIO_RDATA".PC_1_CONNECT.DTYP := "DI";
   "DIO_RDATA".PC_1_CONNECT.INVERT := TRUE;
   "DIO_RDATA".PC_1_EXT_OUT.DTYP := "DI";
   "DIO_RDATA".PC_1_EXT_OUT.INVERT := TRUE;
   "DIO_RDATA".EE_1_FS.DTYP := "DI";
   "DIO_RDATA".EE_1_FS.INVERT := TRUE;
   "DIO_RDATA".POLSW_1_POS1.DTYP := "DI";
   "DIO_RDATA".POLSW_1_POS1.INVERT := TRUE;
   "DIO_RDATA".POLSW_1_POS2.DTYP := "DI";
   "DIO_RDATA".POLSW_1_POS2.INVERT := TRUE;
   "DIO_RDATA".spare_4.DTYP := "DI";
   "DIO_RDATA".KEY1_OK.DTYP := "DI";
   "DIO_RDATA".KEY1_OK.INVERT := TRUE;
   "DIO_RDATA".NO_QUENCH.DTYP := "DI";
   "DIO_RDATA".NO_QUENCH.INVERT := TRUE;
   "DIO_RDATA".DAQ_OK.DTYP := "DI";
   "DIO_RDATA".DAQ_OK.INVERT := TRUE;

   "DIO_RDATA".EE_2_POWER_PERM.DTYP := "DI";
   "DIO_RDATA".EE_2_POWER_PERM.INVERT := TRUE;
   "DIO_RDATA".EE_2_REMOTE.DTYP := "DI";
   "DIO_RDATA".EE_2_REMOTE.INVERT := TRUE;
   "DIO_RDATA"."EE_2_NO_ERROR_CL".DTYP := "DI";
   "DIO_RDATA"."EE_2_NO_ERROR_CL".INVERT := TRUE;
   "DIO_RDATA".EE_2_CLOSED.DTYP := "DI";
   "DIO_RDATA".EE_2_CLOSED.INVERT := TRUE;
   "DIO_RDATA"."spare_2".DTYP := "DI";
   "DIO_RDATA"."spare_2".INVERT := TRUE;
   "DIO_RDATA".EE_2_PC_SPA_OK.DTYP := "DI";
   "DIO_RDATA".EE_2_PC_SPA_OK.INVERT := TRUE;
   "DIO_RDATA".PC_2_POWER_Failure.DTYP := "DI";
   "DIO_RDATA".PC_2_POWER_Failure.INVERT := TRUE;
   "DIO_RDATA".PC_2_CONNECT.DTYP := "DI";
   "DIO_RDATA".PC_2_CONNECT.INVERT := TRUE;
   "DIO_RDATA".PC_2_EXT_OUT.DTYP := "DI";
   "DIO_RDATA".PC_2_EXT_OUT.INVERT := TRUE;
   "DIO_RDATA".EE_2_FS.DTYP := "DI";
   "DIO_RDATA".EE_2_FS.INVERT := TRUE;
   "DIO_RDATA".POLSW_2_POS1.DTYP := "DI";
   "DIO_RDATA".POLSW_2_POS1.INVERT := TRUE;
   "DIO_RDATA".POLSW_2_POS2.DTYP := "DI";
   "DIO_RDATA".POLSW_2_POS2.INVERT := TRUE;
   "DIO_RDATA".spare_8.DTYP := "DI";
   "DIO_RDATA".DC24V_AUX1_OK.DTYP := "DI";
   "DIO_RDATA".DC24V_AUX1_OK.INVERT := TRUE;
   "DIO_RDATA".KEY2_OK.DTYP := "DI";
   "DIO_RDATA".KEY2_OK.INVERT := TRUE;
   "DIO_RDATA".DC24V_AUX2_OK.DTYP := "DI";
   "DIO_RDATA".DC24V_AUX2_OK.INVERT := TRUE;


   // Software DI
   "DIO_RDATA".LEAD_1_TEMP_OK.DTYP := "DI";
   "DIO_RDATA".LEAD_1_TEMP_OK.INVERT := TRUE;
   "DIO_RDATA".LEAD_2_TEMP_OK.DTYP := "DI";
   "DIO_RDATA".LEAD_2_TEMP_OK.INVERT := TRUE;
   "DIO_RDATA".LEAD_3_TEMP_OK.DTYP := "DI";
   "DIO_RDATA".LEAD_3_TEMP_OK.INVERT := TRUE;
   "DIO_RDATA".LEAD_4_TEMP_OK.DTYP := "DI";
   "DIO_RDATA".LEAD_4_TEMP_OK.INVERT := TRUE;
   "DIO_RDATA"."CRYO_1.9K".DTYP := "DI";
   "DIO_RDATA"."CRYO_1.9K".INVERT := TRUE;
   "DIO_RDATA"."CRYO_4.5K".DTYP := "DI";
   "DIO_RDATA"."CRYO_4.5K".INVERT := TRUE;
   "DIO_RDATA".CRYO_300K_HE.DTYP := "DI";
   "DIO_RDATA".CRYO_300K_HE.INVERT := TRUE;
   "DIO_RDATA".CRYO_300K_AIR.DTYP := "DI";
   "DIO_RDATA".CRYO_300K_AIR.INVERT := TRUE;
   "DIO_RDATA".CRYO_LEADS_OK.DTYP := "DI";
   "DIO_RDATA".CRYO_LEADS_OK.INVERT := TRUE;
   "DIO_RDATA".LEAD_1_VOLT_OK.DTYP := "DI";
   "DIO_RDATA".LEAD_1_VOLT_OK.INVERT := TRUE;
   "DIO_RDATA".LEAD_2_VOLT_OK.DTYP := "DI";
   "DIO_RDATA".LEAD_2_VOLT_OK.INVERT := TRUE;
   "DIO_RDATA".LEAD_3_VOLT_OK.DTYP := "DI";
   "DIO_RDATA".LEAD_3_VOLT_OK.INVERT := TRUE;
   "DIO_RDATA".LEAD_4_VOLT_OK.DTYP := "DI";
   "DIO_RDATA".LEAD_4_VOLT_OK.INVERT := TRUE;

   // Hardware DO
   // 

   "DIO_RDATA".EE_1_OPEN_RQ.DTYP := "DO";
   "DIO_RDATA".spare27.DTYP := "DO";
   "DIO_RDATA".spare28.DTYP := "DO";
   "DIO_RDATA".PC_1_PERMIT.DTYP := "DO";
   "DIO_RDATA".PC_1_PERMIT.INVERT := TRUE;
   "DIO_RDATA".PC_1_PERMIT.N_LATCH := TRUE;
   "DIO_RDATA".PC_1_EXT.DTYP := "DO";
   "DIO_RDATA".PC_1_EXT.INVERT := TRUE;
   "DIO_RDATA".PC_1_EXT.N_LATCH := TRUE;
   "DIO_RDATA".spare_9.DTYP := "DO";
   "DIO_RDATA".spare_10.DTYP := "DO";
   "DIO_RDATA".spare_11.DTYP := "DO";
   "DIO_RDATA".spare_3.DTYP := "DO";
   "DIO_RDATA".spare_3.INVERT := TRUE;
   "DIO_RDATA".spare_3.N_LATCH := TRUE;
   "DIO_RDATA".spare31.DTYP := "DO";
   "DIO_RDATA".spare31.N_LATCH := TRUE;
   "DIO_RDATA".spare31.INVERT := TRUE;
   "DIO_RDATA".spare32.DTYP := "DO";
   "DIO_RDATA".spare32.N_LATCH := TRUE;
   "DIO_RDATA".spare33.DTYP := "DO";
   "DIO_RDATA".spare33.N_LATCH := TRUE;
   "DIO_RDATA".spare_12.DTYP := "DO";
   "DIO_RDATA".spare_13.DTYP := "DO";
   "DIO_RDATA".spare_14.DTYP := "DO";
   "DIO_RDATA".spare_15.DTYP := "DO";

   "DIO_RDATA".EE_2_OPEN_RQ.DTYP := "DO";
   "DIO_RDATA".spare29.DTYP := "DO";
   "DIO_RDATA".spare30.DTYP := "DO";
   "DIO_RDATA".PC_2_PERMIT.DTYP := "DO";
   "DIO_RDATA".PC_2_PERMIT.INVERT := TRUE;
   "DIO_RDATA".PC_2_PERMIT.N_LATCH := TRUE;
   "DIO_RDATA".PC_2_EXT.DTYP := "DO";
   "DIO_RDATA".PC_2_EXT.INVERT := TRUE;
   "DIO_RDATA".PC_2_EXT.N_LATCH := TRUE;
   "DIO_RDATA".spare_16.DTYP := "DO";
   "DIO_RDATA".spare_17.DTYP := "DO";
   "DIO_RDATA".spare_18.DTYP := "DO";
   "DIO_RDATA".spare_19.DTYP := "DO";
   "DIO_RDATA".spare_20.DTYP := "DO";
   "DIO_RDATA".spare_21.DTYP := "DO";
   "DIO_RDATA".spare_22.DTYP := "DO";
   "DIO_RDATA".spare_23.DTYP := "DO";
   "DIO_RDATA".spare_24.DTYP := "DO";
   "DIO_RDATA".spare_25.DTYP := "DO";

   //"EE_1_OPEN_RQ" := "DIO_RDATA".EE_1_OPEN_RQ.VAL;
   "CLOSE_EE_1" := "CPU_RDATA".CPU_CONF.EE_1_CLOSE;
   "RESET_EE_1" := "CPU_RDATA".CPU_CONF.EE_1_RESET;
   "PC_1_PERMIT" := "DIO_RDATA".PC_1_PERMIT.VAL;
   "PC_1_EXT" := "DIO_RDATA".PC_1_EXT.VAL;


   // := "DIO_RDATA".spare_3.VAL;

   //"EE_2_OPEN_RQ" := "DIO_RDATA".EE_2_OPEN_RQ.VAL;
   "CLOSE_EE_2" := "CPU_RDATA".CPU_CONF.EE_2_CLOSE;
   "RESET_EE_2" := "CPU_RDATA".CPU_CONF.EE_2_RESET;
   "PC_2_PERMIT" := "DIO_RDATA".PC_2_PERMIT.VAL;
   "PC_2_EXT" := "DIO_RDATA".PC_2_EXT.VAL;


   // The mbi (Marker Binary Output) is being handled by the Machine State
   // 0 = no interlock
   // 1 = Interlock
   ////"DIO_RDATA".FIM_110_HVena.INTERLOCK := "mbo_hvonInterlock";
   ////"DIO_RDATA".FIM_110_RFena.INTERLOCK := "mbo_rfonInterlock";

   ////"FIM_110_HVena":P  := "DIO_RDATA".FIM_110_HVena.VAL;
   ////"FIM_110_RFena":P  := "DIO_RDATA".FIM_110_RFena.VAL;

   // Light indicators

   ////"Kly_110_GreenLight":P := "DIO_RDATA".Kly_110_GreenLight.VAL;

   ////"DA_110_DArst" := "DIO_RDATA".DA_110_DArst.VAL;
   ////"DA_110_DAena" := "DIO_RDATA".DA_110_DAena.VAL;
   //

   ///////////////////////////////////////////////////////////////////////////////////////////
   // Interlock rules
   /////////////////////////////////////////////////////////////////////////////////////////// 

   // Power Converter Permit interlock
   // 

   #POLSW_INTERLOCK_1 := NOT("DIO_RDATA".POLSW_1_POS1.INTERLOCK XOR "DIO_RDATA".POLSW_1_POS2.INTERLOCK);

   "DIO_RDATA".PC_1_PERMIT.INTERLOCK := "DIO_RDATA".NO_QUENCH.INTERLOCK OR
   "DIO_RDATA".KEY1_OK.INTERLOCK OR
   "DIO_RDATA".DAQ_OK.INTERLOCK OR "DIO_RDATA".DC24V_AUX1_OK.INTERLOCK OR
   "DIO_RDATA".DC24V_AUX2_OK.INTERLOCK OR
   "DIO_RDATA".EE_1_CLOSED.INTERLOCK OR "DIO_RDATA".EE_1_NO_ERROR_CL.INTERLOCK OR
   "DIO_RDATA".EE_1_PC_SPA_OK.INTERLOCK OR
   "DIO_RDATA".EE_1_POWER_PERM.INTERLOCK OR "DIO_RDATA".EE_1_REMOTE.INTERLOCK OR
   "DIO_RDATA".LEAD_1_TEMP_OK.INTERLOCK OR "DIO_RDATA".LEAD_2_TEMP_OK.INTERLOCK OR
   "DIO_RDATA".LEAD_1_VOLT_OK.INTERLOCK OR "DIO_RDATA".LEAD_2_VOLT_OK.INTERLOCK OR
   "DIO_RDATA".PC_1_CONNECT.INTERLOCK OR "DIO_RDATA".PC_1_EXT_OUT.INTERLOCK OR
   "DIO_RDATA".PC_1_POWER_Failure.INTERLOCK OR NOT("CPU_RDATA".CPU_CONF.GERSEMI_COM_OK) OR
   "DIO_RDATA".EE_1_FS.INTERLOCK OR #POLSW_INTERLOCK_1;

   #POLSW_INTERLOCK_2 := NOT("DIO_RDATA".POLSW_2_POS1.INTERLOCK XOR "DIO_RDATA".POLSW_2_POS2.INTERLOCK);

   "DIO_RDATA".PC_2_PERMIT.INTERLOCK := "DIO_RDATA".NO_QUENCH.INTERLOCK OR
   "DIO_RDATA".KEY2_OK.INTERLOCK OR
   "DIO_RDATA".DAQ_OK.INTERLOCK OR "DIO_RDATA".DC24V_AUX1_OK.INTERLOCK OR
   "DIO_RDATA".DC24V_AUX2_OK.INTERLOCK OR
   "DIO_RDATA".EE_2_CLOSED.INTERLOCK OR "DIO_RDATA".EE_2_NO_ERROR_CL.INTERLOCK OR
   "DIO_RDATA".EE_2_PC_SPA_OK.INTERLOCK OR
   "DIO_RDATA".EE_2_POWER_PERM.INTERLOCK OR "DIO_RDATA".EE_2_REMOTE.INTERLOCK OR
   "DIO_RDATA".LEAD_3_TEMP_OK.INTERLOCK OR "DIO_RDATA".LEAD_4_TEMP_OK.INTERLOCK OR
   "DIO_RDATA".LEAD_3_VOLT_OK.INTERLOCK OR "DIO_RDATA".LEAD_4_VOLT_OK.INTERLOCK OR
   "DIO_RDATA".PC_2_CONNECT.INTERLOCK OR "DIO_RDATA".PC_2_EXT_OUT.INTERLOCK OR
   "DIO_RDATA".PC_2_POWER_Failure.INTERLOCK OR NOT("CPU_RDATA".CPU_CONF.GERSEMI_COM_OK) OR
   "DIO_RDATA".EE_2_FS.INTERLOCK OR #POLSW_INTERLOCK_1;

   // Direct Power Abort Interlock
   // 

   // Fast power abort
   // 
   "DIO_RDATA".PC_1_EXT.INTERLOCK := "DIO_RDATA".KEY1_OK.INTERLOCK OR
   "DIO_RDATA".DC24V_AUX1_OK.INTERLOCK OR "DIO_RDATA".DC24V_AUX2_OK.INTERLOCK OR
   "DIO_RDATA".NO_QUENCH.INTERLOCK OR #POLSW_INTERLOCK_1;

   "DIO_RDATA".PC_2_EXT.INTERLOCK := "DIO_RDATA".KEY2_OK.INTERLOCK OR
   "DIO_RDATA".DC24V_AUX1_OK.INTERLOCK OR "DIO_RDATA".DC24V_AUX2_OK.INTERLOCK OR
   "DIO_RDATA".NO_QUENCH.INTERLOCK OR #POLSW_INTERLOCK_2;

   // EE open request
   // 
   "IEC_Timer_EE1_DB".TP(IN:="DIO_RDATA".PC_1_EXT.INTERLOCK,
                       PT:=#pulse_time,
                       Q=>#EE_1_Open_RQ,
                       ET=>#t1);
   "EE_1_OPEN_RQ" := NOT(#EE_1_Open_RQ);

   "IEC_Timer_EE2_DB".TP(IN:="DIO_RDATA".PC_2_EXT.INTERLOCK,
                         PT:=#pulse_time,
                         Q=>#EE_2_Open_RQ,
                         ET=>#t2);
   "EE_2_OPEN_RQ" := NOT (#EE_2_Open_RQ);


   // Flash lights
   //
   "CPU_RDATA".CPU_CONF.FLSHBX_HV := NOT  ("DIO_RDATA".PC_1_EXT_OUT.INTERLOCK AND "DIO_RDATA".PC_2_EXT_OUT.INTERLOCK);
   "FLSHBX_HVOLT" := "CPU_RDATA".CPU_CONF.FLSHBX_HV;

   "CPU_RDATA".CPU_CONF.FLSHBX_HC := NOT ("DIO_RDATA".PC_1_EXT_OUT.INTERLOCK AND "DIO_RDATA".PC_2_EXT_OUT.INTERLOCK);
   "FLSHBX_HCUR" := "CPU_RDATA".CPU_CONF.FLSHBX_HC;

   "CPU_RDATA".CPU_CONF.FLSHBX_He := NOT ("DIO_RDATA".PC_1_PERMIT.INTERLOCK AND "DIO_RDATA".PC_2_PERMIT.INTERLOCK);
   "FLSHBX_HE" := "CPU_RDATA".CPU_CONF.FLSHBX_He;

   //"AI00_AMP" := INT_TO_REAL("KLY_Oil_FSn_WatOutletFlow") * 16.0 / 27648.0 + 4.0; (*basic convertion to mAMPS*)
END_FUNCTION

ORGANIZATION_BLOCK "Main"   // OB1, SCL, ProgramCycle
TITLE = Program cycle
{ S7_Optimized_Access := 'FALSE' }
VERSION : 0.1
   VAR_TEMP
      EV_CLASS : Byte;   // Bits 0-3 = 1:Coming event, Bits 4-7 = 1:Event class 1
      SCAN_1 : Byte;   // 1:Initial call of the OB, 3: Call 2-n of the OB
      PRIORITY : Byte;   // Priority of OB Execution
      OB_NUMBR : Byte;   // OB number
      RESERVED_1 : Byte;   // Reserved for system
      RESERVED_2 : Byte;   // Reserved for system
      PREV_CYCLE : Int;   // Previous program cycle time (milliseconds)
      MIN_CYCLE : Int;   // Minimum program cycle time (milliseconds)
      MAX_CYCLE : Int;   // Maximum program cycle time (milliseconds)
      DATE_TIME : Date_And_Time;   // Date and time OB started
   END_VAR
BEGIN
   // Send receive communication function
   // --> EPICS_Communication Group folder
   "Send_Receive"();

   //Get the field values from the IO module
   "GET_MEASUREMENT"();

   // This function contains the IO signal processing
   // --> SignalProcessing Group folder
   "CHKVARS"();

   // This function contains the communication with Gesremi PLC
   // --> Gersemi_Communication Group folder
   "Gersemi_Com"();

   // Get Operation Location
   // To be implemented with the Local/Remote key
   // "GET_LOCATION"(LOCATION:= "Remote_SwPos",
   //               LOCATION => "mb_location");

   // Set new Amplifier State
   // According to the Key status, the amplifier can be controlled locally or remotely
   ////"SET_AMP_STATE"(CPU_CONF:="CPU_RDATA".CPU_CONF,
   ////                SET_STATE:= "mw_setState");

   // Function required to get the Timestamp, but it can be replaced
   // or processed internally into the AF_ and DIO_ "Signal processing"
   "TD_TO_INT"();

   // Main LPS logic and Machine State operation GRAPH
   // --> MachineState Group folder
   ////"STATE_MACHINE_DB"(INIT_SQ := True);
END_ORGANIZATION_BLOCK

ORGANIZATION_BLOCK "COMPLETE RESTART"   // OB100, SCL, Startup
TITLE = "Complete Restart"
{ S7_Optimized_Access := 'FALSE' }
VERSION : 0.1
   VAR_TEMP
      OB100_EV_CLASS : Byte;   // 16#13, Event class 1, Entering event state, Event logged in diagnostic buffer
      OB100_STRTUP : Byte;   // 16#81/82/83/84 Method of startup
      OB100_PRIORITY : Byte;   // Priority of OB Execution
      OB100_OB_NUMBR : Byte;   // 100 (Organization block 100, OB100)
      OB100_RESERVED_1 : Byte;   // Reserved for system
      OB100_RESERVED_2 : Byte;   // Reserved for system
      OB100_STOP : Word;   // Event that caused CPU to stop (16#4xxx)
      OB100_STRT_INFO : DWord;   // Information on how system started
      OB100_DATE_TIME : Date_And_Time;   // Date and time OB100 started
   END_VAR
BEGIN
   //datain_TCP1.CPU_STATUS.STAT := 2;
   //"dataout_TCP1".CPU_STATUS.STAT := W#16#2;
   //"CPU_RDATA".CPU_STATUS.STAT := W#16#02;

   //"CPU_RDATA".CPU_CONF.OP_MODE := #OB100_STRTUP;

   //New device type parametrisation
   //

   "TCP1_instance"(INIT_COM := True,                             // IN: BOOL
                   RECV_DB := "CPU_WDATA",
                   SEND_DB := "CPU_RDATA",
                   C_PARAM := "CH_PARAM_TCP_CPU".CommParam);     // IN_OUT: STRUCT

   "TCP2_instance"(INIT_COM := True,                             // IN: BOOL
                   RECV_DB := "AF_WDATA",
                   SEND_DB := "AF_RDATA",
                   C_PARAM := "CH_PARAM_TCP_AF".CommParam);     // IN_OUT: STRUCT

   "TCP3_instance"(INIT_COM:=TRUE,
                   RECV_DB:="DIO_WDATA",
                   SEND_DB:="DIO_RDATA",
                   C_PARAM:="CH_PARAM_TCP_DIO".CommParam);

   "TCP4_instance"(INIT_COM := True,                             // IN: BOOL
                   RECV_DB := "PSU_WDATA",
                   SEND_DB := "PSU_RDATA",
                   C_PARAM := "CH_PARAM_TCP_PSU".CommParam);     // IN_OUT: STRUCT

   // "AF_RDATA".KLY_SOL_SURF_TP.DTYP := "TSn";
   // "AF_RDATA".KLY_SOL_WAT_INLET_FM.DTYP := "TSn";
   // "AF_RDATA".KLY_SOL_WAT_INLET_TP.DTYP := "VSn_0_10v";

   // "DIO_RDATA".RFS_RF_ENABLE_DO.DTYP := "DO";
   // "DIO_RDATA".RFS_HV_ENABLE_DO.DTYP := "DO";

   "CPU_RDATA".CPU_CONF.LATCH_MODE := True;

   "InstDiagStartupPlc"(plc := "DiagnosticsData".plc);

   //
   //We do not have PROFINET IO system
   ////"InstDiagStartupIoSystem"(ioSystemHwId:="Local~PROFINET_IO-System",
   //                          ioSystem:="DiagnosticsData".ioSystem["IO_SYSTEM1"]);
END_ORGANIZATION_BLOCK

// folder: Diagnostics

FUNCTION_BLOCK "Diagnostics"   // FB2000, SCL
{ S7_Optimized_Access := 'TRUE' }
VERSION : 0.1
   VAR_INPUT
      firstCyleInit : Bool := TRUE;   // in first cycle TRUE
   END_VAR
   VAR_IN_OUT
      plc : "typePlc";   // The diagnostics structure for one PLC
      showPlc : "typeShowPlc";   // The show diagnostics structure for one PLC
      ioSystem : Array[1.."MAX_SYSTEM"] of "typeIoSystem";   // The diagnostics structure for one IO System
      showIoSystem : Array[1.."MAX_SYSTEM"] of "typeShowIoSystem";   // The show diagnostics structure for one IO System
      showActIoSystem : "typeShowActIoSystem";   // The show diagnostics structure for the selected IO System
   END_VAR
   VAR
      statIoSystemIndex : Int;   // Index for IO System
      statSlotIndex : Int;   // Index for Slot
      statDeviceIndex : Int;   // Index for Device
   END_VAR
   VAR_TEMP
      retValLed : Int;
   END_VAR
   VAR CONSTANT
      ERROR_LED : UInt := 2;   // Identification number of the ERROR LED
      ERROR_LED_ON : UInt := 4;   // LED status Color 1 flashing
   END_VAR
BEGIN
   //=============================================================================
   //SIEMENS AG
   //(c)Copyright 2015 All Rights Reserved
   //-----------------------------------------------------------------------------
   //Library: -
   //Tested with: S7-1516-3 PN/DP FW 1.7
   //Engineering: TIA Portal V13 SP1
   //Restrictions: -
   //Requirements: -
   //Functionality: copy and control diagnosis information for visualization
   //-----------------------------------------------------------------------------
   //Change log table:
   //Version  Date       Expert in charge Changes applied
   //01.00.00 24.03.2015 Siemens Industry Online Support First released version
   //=============================================================================

   //=============================================================================
   // copy diagnosis information to ShowDiag DB for visualization in first cycle
   //=============================================================================
   IF (#firstCyleInit = TRUE)
   THEN
     // copy PLC diagnosis information to ShowDiag DB 
     #showPlc.errorState := #plc.errorState;
     FOR #statSlotIndex := 1 TO "MAX_MODULES_LOCAL" DO

       IF #plc.slot[#statSlotIndex].slotLaddr <> 0
       THEN
         #showPlc.slot[#statSlotIndex].slotErrorState := #plc.slot[#statSlotIndex].slotErrorState;
         #showPlc.slot[#statSlotIndex].slotUsed := TRUE;
       ELSE
         #showPlc.slot[#statSlotIndex].slotUsed := FALSE;
       END_IF;
     END_FOR;

     // copy device diagnosis information for each IO system to "ShowDiag" DB
     FOR #statIoSystemIndex := 1 TO "MAX_SYSTEM" DO

       FOR #statDeviceIndex := 1 TO "MAX_DEVICES_SYSTEM" DO
         #showIoSystem[#statIoSystemIndex].device[#statDeviceIndex].stationNumber := INT_TO_UINT(#statDeviceIndex);
         #showIoSystem[#statIoSystemIndex].device[#statDeviceIndex].name := #ioSystem[#statIoSystemIndex].device[#statDeviceIndex].name;
         #showIoSystem[#statIoSystemIndex].device[#statDeviceIndex].errorState := #ioSystem[#statIoSystemIndex].device[#statDeviceIndex].errorState;

         FOR #statSlotIndex := 0 TO "MAX_MODULES_DEVICE" DO

           IF (#ioSystem[#statIoSystemIndex].device[#statDeviceIndex].slot[#statSlotIndex].slotLaddr <> 0)
           THEN
             #showIoSystem[#statIoSystemIndex].device[#statDeviceIndex].slot[#statSlotIndex].slotErrorState := #ioSystem[#statIoSystemIndex].device[#statDeviceIndex].slot[#statSlotIndex].slotErrorState;
             #showIoSystem[#statIoSystemIndex].device[#statDeviceIndex].slot[#statSlotIndex].slotUsed := TRUE;
           ELSE
             #showIoSystem[#statIoSystemIndex].device[#statDeviceIndex].slot[#statSlotIndex].slotUsed := FALSE;
           END_IF;
         END_FOR;
       END_FOR;

     END_FOR;

   END_IF;



   //=============================================================================
   // check error active
   //=============================================================================
   #retValLed := LED(LADDR := "Local~Common", LED := #ERROR_LED);
   IF #retValLed = #ERROR_LED_ON
   THEN
     #plc.errorState := TRUE;
   ELSE
     #plc.errorState := FALSE;
   END_IF;

   //=============================================================================
   // check error in IO systems active
   //=============================================================================
   FOR #statIoSystemIndex := 1 TO "MAX_SYSTEM" DO
     #ioSystem[#statIoSystemIndex].ioSystemError := FALSE;

     FOR #statDeviceIndex := 1 TO "MAX_DEVICES_SYSTEM" DO
       IF (#ioSystem[#statIoSystemIndex].device[#statDeviceIndex].error = TRUE)
       THEN
         #ioSystem[#statIoSystemIndex].ioSystemError := TRUE;
       END_IF;
     END_FOR;
   END_FOR;


   //=============================================================================
   // HMI control
   //=============================================================================

   //=============================================================================
   // check index of IO system from HMI
   //=============================================================================
   IF (#showActIoSystem.actIoSystem > "MAX_SYSTEM")
   THEN
     #showActIoSystem.actIoSystem := "MAX_SYSTEM";
   END_IF;

   //=============================================================================
   // copy diagnosis information to PLC for visualization
   //=============================================================================
   IF (#showPlc.diagnosisLoaded = TRUE)
   THEN
     #showPlc.errorState := #plc.errorState;
   //  #showPlc.diagnosisLoaded := FALSE;
   ELSE
     ;// No initialization needed
   END_IF;

   //=============================================================================
   // copy diagnosis information to active IO system for visualization
   //=============================================================================
   IF (#showActIoSystem.diagnosisLoaded = TRUE)
   THEN
     #showActIoSystem.device := #showIoSystem[#showActIoSystem.actIoSystem].device;
     #showActIoSystem.diagnosisLoaded := FALSE;
   ELSE
     ;// No initialization needed
   END_IF;

   //=============================================================================
   // copy device state of the selected device in HMI to active device
   // to show the module state
   //=============================================================================
   IF (#showActIoSystem.copyModuleStates = TRUE)
   THEN
     #showActIoSystem.actDevice := #showIoSystem[#showActIoSystem.actIoSystem].device[#showActIoSystem.actDeviceIndex];
   END_IF;

   //=============================================================================
   // Reset "was faulty" and "was lost" devices and slaves to "ok!"
   //=============================================================================

   // Detect a rising edge at ResetStates and start initializing
   IF (#showActIoSystem.resetStates = TRUE)
   THEN
     // Reset PN Devices
     FOR #statDeviceIndex := 1 TO "MAX_DEVICES_SYSTEM" DO
       IF ((#ioSystem[#showActIoSystem.actIoSystem].device[#statDeviceIndex].errorState = "DEV_STATE_WAS_FAULT") OR
           (#ioSystem[#showActIoSystem.actIoSystem].device[#statDeviceIndex].errorState = "DEV_STATE_WAS_LOST") OR
           (#ioSystem[#showActIoSystem.actIoSystem].device[#statDeviceIndex].errorState = "DEV_STATE_WAS_DISABLED"))
       THEN
         #ioSystem[#showActIoSystem.actIoSystem].device[#statDeviceIndex].errorState := "DEV_STATE_OK";
         #ioSystem[#showActIoSystem.actIoSystem].device[#statDeviceIndex].error := FALSE;

         // copy diagnosis information to ShowDiag DB
         "CopyToHmiDB"(deviceIndex := #statDeviceIndex,
                       plc := #plc,
                       showPlc := #showPlc,
                       ioSystem := #ioSystem[#showActIoSystem.actIoSystem],
                       showIoSystem := #showIoSystem[#showActIoSystem.actIoSystem]);

       ELSE
         ;
       END_IF;
     END_FOR;

     // update visualization
     #showActIoSystem.device := #showIoSystem[#showActIoSystem.actIoSystem].device;

   ELSE
     ;// No initialization needed
   END_IF;
END_FUNCTION_BLOCK

FUNCTION_BLOCK "DiagStartupIoSystem"   // FB2001, SCL
{ S7_Optimized_Access := 'TRUE' }
VERSION : 0.1
   VAR_INPUT
      ioSystemHwId : Hw_IoSystem;   // This ID is representing the IO System (PN or DP), find the ID in the system constants
   END_VAR
   VAR_OUTPUT
      status : Int;   // The return value of system function, where the last error occured
      instructionError : Int;   // Indicates in which system function the error occured: 1= DeviceStates PN , 2=GetName PN, 3=ModuleStates PN, 4=DeviceStates DP, 5= GetName DP. 6= ModuleStates DP
      errorIndex : Int;   // The last index of the respective loop, if an error occures
   END_VAR
   VAR_IN_OUT
      ioSystem : "typeIoSystem";   // The diagnostics structure for one IO System
   END_VAR
   VAR
      statActualConfiguredDevices : Int := 0;   // Actual number of devices in the PN IO System
      statGeoAddr : GEOADDR;   // Slot information
      statGeoLaddr : Hw_Any;   // GEO2LOG hardware identifier
      statConfiguredDevices : Array[0..1023] of Bool;   // Temporary storage of the return of "DeviceStates", to combine the states of the devices with numbers and names
      statExistingDevices : Array[0..1023] of Bool;   // Temporary storage of the return of "DeviceStates", to combine the states of the devices with numbers and names
      statFaultyDevices : Array[0..1023] of Bool;   // Temporary storage of the return of "DeviceStates", to combine the states of the divices with numbers and names
      statDisabledDevices : Array[0..1023] of Bool;   // Storage of the status of all devices in the PN IO System --> State: Disabled
      statProblemDevices : Array[0..1023] of Bool;   // Storage of the status of all devices in the PN IO System --> State: Problem
      statDeviceModuleStates : Array[0..127] of Bool;   // Storage of the status of all modules in the PN Devices --> State: Problem
      instGetNameDevices : Get_Name;   // Instance of system function "GetName"
      statInitString : String;   // Used to initialize the temporary string to convert into STRING[50]
      statFirstDevice : UInt;   // Station number of the first device of the list
      statFirstDeviceFlag : Bool := TRUE;   // Help tag for the first device in the linked list
      statLastDevice : UInt;   // Station number of the last device of the list
      statLinkedListPointer : Int;   // The actual index pointer of the linked list (Actual pointer = Station number of the device)
      statFirstRun : Bool := TRUE;   // Signalizes the first run
      statResetStatesOld : Bool;   // Detect a rising edge at ResetStates
      statMaxDevices : Int;
   END_VAR
   VAR_TEMP
      tempIndex : Int;   // index configured devices
      tempSlotIndex : Int;   // Loop index
      tempModuleNum : Int;   // index module number
      tempRetValGeo : Int;   // GEO2LOG error information
      tempRetValDeviceStates : Int;   // DeviceStates error information
      tempRetValModuleStates : Int;   // Return value system function ModuleStates
      tempStringConvert : String;   // Store the device names temporary here, to convert them into STRING[50]
      tempLastDevice : UInt;   // Temporary storage of the actual index, if it´s the last device --> store it in static
      tempIoSystemError : Bool;
   END_VAR
   VAR CONSTANT
      STATE_CONFIGURED : USInt := 1;   // Used for instruction DeviceStates, read out all configured devices
      STATE_FAULTY : USInt := 2;   // Used for instruction DeviceStates, read out all faulty devices
      STATE_DISABLED : USInt := 3;   // Used for instruction DeviceStates, read out all disabled devices
      STATE_EXIST : USInt := 4;   // Used for instruction DeviceStates, read out all devices not reachable
      STATE_PROBLEM : USInt := 5;   // Used for instruction DeviceStates, read out all devices with several problems
      DEVICE_SLAVE : USInt := 2;   // GEO2LOG structure: HW type = 2
      MODULE_OF_DEVICE : USInt := 4;   // GEO2LOG structure: HW type = 4
      IO_SYSTEM_AREA : USInt := 1;   // GEO2LOG structure: Area = 1
      DP_SYSTEM_AREA : USInt := 2;   // GEO2LOG structure: Area = 2
      ERR_DEV_STATE_DEVICES : USInt := 1;   // Identifies the instruction behind the error code of output "Status" --> DeviceStates PN (Configured, faulty, existing)
      ERR_GET_NAME_DEVICES : USInt := 2;   // Identifies the instruction behind the error code of output "Status" --> GetName of devices PN
      ERR_MOD_STAT_DEVICES : USInt := 3;   // Identifies the instruction behind the error code of output "Status" --> ModuleStates PN
      ERR_DEV_STAT_PN : USInt := 1;   // Value for output instruction error, DeviceStates PN devices
      ERR_MOD_STAT_PN : USInt := 4;   // Value for output instruction error, ModuleStates PN devices
      MAX_SLAVES_DP : Int := 127;
   END_VAR
BEGIN
   //=============================================================================
   //SIEMENS AG
   //(c)Copyright 2015 All Rights Reserved
   //-----------------------------------------------------------------------------
   //Library: -
   //Tested with: S7-1516-3 PN/DP FW 1.7
   //Engineering: TIA Portal V13 SP1
   //Restrictions: -
   //Requirements: -
   //Functionality: Determine hardware identifier and module states from devices
   //-----------------------------------------------------------------------------
   //Change log table:
   //Version  Date       Expert in charge Changes applied
   //01.00.00 24.03.2015 Siemens Industry Online Support First released version
   //=============================================================================

   // The startup will be executed only once --> initialize the first run
   // indicator.
   #statFirstDeviceFlag := TRUE;
   #statFirstRun := TRUE;
   #statActualConfiguredDevices := 0;
   #statFirstDevice := 1;
   #statLastDevice := 1;

   //=============================================================================
   // CONFIGURED DEVICES
   //=============================================================================
   // Find out how much devices are configured in the IO System --> PROFINET IO
   // This number is the maximum number of devices, which will be checked in the
   // following programm
   #tempRetValDeviceStates := DeviceStates(LADDR := #ioSystemHwId,
                                           MODE := #STATE_CONFIGURED,
                                           STATE := #statConfiguredDevices);

   // Check if the block call was successful
   IF (#tempRetValDeviceStates <> 0)
   THEN
     // Error handling
     #status := #tempRetValDeviceStates;
     #instructionError := #ERR_DEV_STATE_DEVICES;
     // Call ok --> store the actual number of configured devices    
   ELSE
     ;
   END_IF;

   //=============================================================================
   // EXISTING DEVICES
   //=============================================================================
   #tempRetValDeviceStates := DeviceStates(LADDR := #ioSystemHwId,
                                           MODE := #STATE_EXIST,
                                           STATE := #statExistingDevices);

   // Check if the block call was successful
   IF (#tempRetValDeviceStates <> 0)
   THEN
     // Error handling
     #status := #tempRetValDeviceStates;
     #instructionError := #ERR_DEV_STATE_DEVICES;
     // Call ok --> store the actual number of configured devices    
   ELSE
     ;
   END_IF;

   //=============================================================================
   // FAULTY DEVICES
   //=============================================================================
   #tempRetValDeviceStates := DeviceStates(LADDR := #ioSystemHwId,
                                           MODE := #STATE_FAULTY,
                                           STATE := #statFaultyDevices);

   // Check if the block call was successful
   IF (#tempRetValDeviceStates <> 0)
   THEN
     // Error handling
     #status := #tempRetValDeviceStates;
     #instructionError := #ERR_DEV_STATE_DEVICES;
     // Call ok --> store the actual number of configured devices    
   ELSE
     ;
   END_IF;

   // Find out the number of the assigned IO system, to define if it is
   // a PN or DP Network
   #tempRetValGeo := LOG2GEO(LADDR := #ioSystemHwId,
                             GEOADDR := #statGeoAddr);

   // set IO system ID
   #ioSystem.ioSystemId := #statGeoAddr.IOSYSTEM;

   // Inilize the structure for system function GEO2LOG
   #statGeoAddr.HWTYPE := #DEVICE_SLAVE;   // Hardware type 2: IO device
   // Predefine the type OF IO system. Either Profinet IO or Profibus DP
   IF ((#statGeoAddr.IOSYSTEM >= 100) 
     AND (#statGeoAddr.IOSYSTEM <= 115))
   THEN
     #statGeoAddr.AREA := #IO_SYSTEM_AREA;   // Area ID 1: PROFINET IO
     #statMaxDevices := "MAX_DEVICES_SYSTEM";
   ELSIF ((#statGeoAddr.IOSYSTEM >= 1)
     AND (#statGeoAddr.IOSYSTEM <= 32))
   THEN
     #statGeoAddr.AREA := #DP_SYSTEM_AREA;   // Area ID 1: Profibus DP
     #statMaxDevices := #MAX_SLAVES_DP;
   ELSE
     ;
   END_IF;

   // Go trough all devices and get the status of the configured
   FOR #tempIndex := 1 TO #statMaxDevices DO
     // The devices are configured --> Read out the logical address and the
     // device name
     IF (#statConfiguredDevices[#tempIndex] = TRUE)
     THEN
       // Increment the actual configured devices, store the state and
       // HW_ID as an numerical value (UINT)
       #statActualConfiguredDevices := #statActualConfiguredDevices + 1;

       // Store the first configured device for the linked list
       IF (#statFirstDeviceFlag = TRUE)
       THEN
         #statFirstDevice := INT_TO_UINT(#tempIndex);
         #ioSystem.firstDevice := UINT_TO_INT(#statFirstDevice);
         #statFirstDeviceFlag := FALSE;
         #tempLastDevice := INT_TO_UINT(#tempIndex);
         // It´s not the first bit --> Store the actual index as "next device"
         // in the further one!
       ELSE
         #ioSystem.device[#tempLastDevice].nextDevice := #tempIndex;
         #tempLastDevice := INT_TO_UINT(#tempIndex);
       END_IF;
       // Store the index of the last device for the exit condition of the
       // followiing instructions
       #statLastDevice := #tempLastDevice;
       #ioSystem.lastDevice := UINT_TO_INT(#statLastDevice);

       // Station number 
       #statGeoAddr.STATION := INT_TO_UINT(#tempIndex);
       // read LADDR from devices
       #tempRetValGeo := GEO2LOG(GEOADDR := #statGeoAddr,
                                 LADDR => #statGeoLaddr);
       // Everything is ok!
       IF (#tempRetValGeo = 0)
       THEN
         // store LADDR from devices in diagnostic data block
         #ioSystem.device[#tempIndex].laddr := #statGeoLaddr;

         // Store the device name, if the device is existing
         // Get name is an acyclic instruction. In the startup OB, the
         // instruction has to be repeated until it is done or error
         REPEAT
           // Get device name of each decive in PN System
           #instGetNameDevices(LADDR := #ioSystemHwId,
                               STATION_NR := #statGeoAddr.STATION,
                               DATA := #tempStringConvert);

         UNTIL (#instGetNameDevices.DONE = TRUE)
           OR (#instGetNameDevices.ERROR = TRUE)
         END_REPEAT;

         IF (#instGetNameDevices.ERROR = TRUE)
         THEN
           // Error handling
           #status := WORD_TO_INT(#instGetNameDevices.STATUS);
           #instructionError := #ERR_GET_NAME_DEVICES;
           #errorIndex := #tempIndex;

           // Everything is ok --> Convert the String[254] into String[50]    
         ELSIF (#instGetNameDevices.DONE = TRUE)
         THEN
           // Cut all characters more than 50 to reduce the string length
           #ioSystem.device[#tempIndex].name := DELETE(IN := #tempStringConvert,
                                                       L := 204,
                                                       P := 50);

           // Initialize the temporary string before next loop
           #tempStringConvert := #statInitString;
         ELSE
           ;
         END_IF;
       ELSE
         // If the return value ist not = 0 --> the device/system/module is
         // not configured --> No error handling
         // set LADDR from devices to 0 in diagnostic data block
         #ioSystem.device[#tempIndex].laddr := 0;
         #ioSystem.device[#tempIndex].name := '';
       END_IF;

       // Check if the configured devices are faulty or lost once through
       // the startup!
       IF (#statExistingDevices[#tempIndex] = TRUE)
       THEN
         IF (#statFaultyDevices[#tempIndex] = TRUE)
         THEN

           #ioSystem.device[#tempIndex].errorState := "DEV_STATE_FAULT";
           #ioSystem.device[#tempIndex].error := TRUE;

           // The device is not faulty and does exist --> set state ok!    
         ELSE
           #ioSystem.device[#tempIndex].errorState := "DEV_STATE_OK";
           #ioSystem.device[#tempIndex].error := FALSE;
         END_IF;
         // The connection to the device is lost at the moment    
       ELSE
         #ioSystem.device[#tempIndex].errorState := "DEV_STATE_LOST_CON";
         #ioSystem.device[#tempIndex].error := TRUE;
       END_IF;
       // No device is configured   
     ELSE
       ;
     END_IF;

   END_FOR;
   // Store the actual configured devices in the diagnostics structure
   #ioSystem.actualConfiguredDevices := #statActualConfiguredDevices;

   // Mark parameter "Next Device" of the last device in the list
   // --> "Next Device" = negative --> Last device in the list
   #ioSystem.device[#statLastDevice].nextDevice := "LAST_DEVICE";

   // Go through the devices until the last device is reached
   // If there are gaps between the device-list, jump over and have a look on
   // the "NextDevice" parameter
   REPEAT
     IF (#statFirstRun = TRUE)
     THEN
       // The index of the linked list is representing the station number.
       #statGeoAddr.STATION := #statFirstDevice;
       // Initialize the pointer for the first run 
       #statLinkedListPointer := UINT_TO_INT(#statFirstDevice);
       // Reset the flag, which signalizes the first run.
       #statFirstRun := FALSE;
     ELSE
       // The index of the linked list is representing the station number.
       #statGeoAddr.STATION := INT_TO_UINT(#statLinkedListPointer);
     END_IF;

     //=============================================================================
     // Get the logical address of all modules and store the actual number of
     // modules from each device
     //=============================================================================

     // Inilize the structure for system function GEO2LOG
     #statGeoAddr.HWTYPE := #MODULE_OF_DEVICE;   // Hardware type 4: Module
     FOR #tempModuleNum := 0 TO "MAX_MODULES_DEVICE" DO
       // Slot number
       #statGeoAddr.SLOT := INT_TO_UINT(#tempModuleNum);
       // read LADDR from modules
       #tempRetValGeo := GEO2LOG(GEOADDR := #statGeoAddr,
                                 LADDR => #statGeoLaddr);
       // check Retval
       IF (#tempRetValGeo = 0)
       THEN
         // store LADDR from modules in diagnostic data block
         #ioSystem.device[#statLinkedListPointer].slot[#tempModuleNum].slotLaddr := #statGeoLaddr;
         #ioSystem.device[#statLinkedListPointer].actualConfiguredModules := #ioSystem.device[#statLinkedListPointer].actualConfiguredModules + 1;
       ELSE
         // If the return value ist not = 0 --> the device/system/module is
         // not configured --> No error handling
         // set LADDR from modules to 0 in diagnostic data block
         #ioSystem.device[#statLinkedListPointer].slot[#tempModuleNum].slotLaddr := 0;
       END_IF;
     END_FOR;

     //=============================================================================
     // Check modules of faulty Devices
     //=============================================================================

     // Check the state of the configured devices
     IF (#ioSystem.device[#statLinkedListPointer].errorState = "DEV_STATE_FAULT")
     THEN
       // The device is reachable, but faulty because of an error in a
       // subordinated system --> check the modules
       #tempRetValModuleStates := ModuleStates(LADDR := #ioSystem.device[#statLinkedListPointer].laddr,
                                               MODE := #STATE_PROBLEM,
                                               STATE := #statDeviceModuleStates);

       IF (#tempRetValModuleStates <> 0)
       THEN
         // Error hanlding
         #status := #tempRetValModuleStates;
         #instructionError := #ERR_MOD_STAT_DEVICES;
         #errorIndex := UINT_TO_INT(#statFirstDevice);
       ELSE
         // Store the state of the different module in the diag DB
         FOR #tempSlotIndex := 0 TO #ioSystem.device[#statFirstDevice].actualConfiguredModules DO
           IF (#statDeviceModuleStates[#tempSlotIndex + 1] = TRUE)
           THEN
             #ioSystem.device[#statLinkedListPointer].slot[#tempSlotIndex].slotErrorState := TRUE;
           ELSE
             #ioSystem.device[#statLinkedListPointer].slot[#tempSlotIndex].slotErrorState := FALSE;
           END_IF;
         END_FOR;
       END_IF;
     ELSIF (#ioSystem.device[#statLinkedListPointer].errorState = "DEV_STATE_LOST_CON")
     THEN

       FOR #tempSlotIndex := 0 TO #ioSystem.device[#statLinkedListPointer].actualConfiguredModules DO
         IF (#ioSystem.device[#statLinkedListPointer].slot[#tempSlotIndex].slotLaddr <> 0)
         THEN
           #ioSystem.device[#statLinkedListPointer].slot[#tempSlotIndex].slotErrorState := TRUE;
         END_IF;
       END_FOR;

     ELSE
       ; // no faulty device --> nothing to do!
     END_IF;

     // Initialize the pointer for the next run
     #statLinkedListPointer := #ioSystem.device[#statLinkedListPointer].nextDevice;
     // If the last device is reached, reset the bit for the first run
     //#FirstRun := TRUE;
     // Checking the modules is done, the last device is reached
   UNTIL (#statLinkedListPointer < 0)
   END_REPEAT;
   // Reset the condition for the first run.
   #statFirstRun := TRUE;
END_FUNCTION_BLOCK

FUNCTION_BLOCK "DiagStartupPlc"   // FB2002, SCL
{ S7_Optimized_Access := 'TRUE' }
VERSION : 0.1
   VAR_OUTPUT
      status : Int;   // The return value of system function, where the last error occured
      instructionError : Int;   // Indicates in which system function the error occured: 1= DeviceStates PN , 2=GetName PN, 3=ModuleStates PN, 4=DeviceStates DP, 5= GetName DP. 6= ModuleStates DP
   END_VAR
   VAR_IN_OUT
      plc : "typePlc";   // The diagnostics structure for one PLC
   END_VAR
   VAR
      statGeoAddr : GEOADDR;   // Slot information
      statGeoLaddr : Hw_Any;   // GEO2LOG hardware identifier
      statActualCentralModules : USInt := 0;   // Actual number of modules in the central station (PLC)
      statPlcModuleStates : Array[0..127] of Bool;   // Storage of the status of all modules in the PLC central station --> State: Problem
   END_VAR
   VAR_TEMP
      tempModuleNum : Int;   // index module number
      tempRetValGeo : Int;   // GEO2LOG error information
      tempRetValModuleStates : Int;   // Return value system function ModuleStates
   END_VAR
   VAR CONSTANT
      MODULE_OF_PLC : USInt := 4;   // GEO2LOG structure: HW type = 4
      CPU : USInt := 0;   // GEO2LOG structure: Area = 0
      CENTRAL_SYSTEM : USInt := 0;   // GEO2LOG structure: IO System = 0
      CENTRAL_STATION : USInt;   // GEO2LOG structure: Station = 0
      HW_ID_PLC_MODULES : Hw_Device := 32;   // HW ID of the PLC, which is needed for getting the module states --> fix value
      STATE_PROBLEM : USInt := 5;   // Used for instruction DeviceStates, read out all devices with several problems
      ERR_MOD_STAT_CENTRAL : USInt := 3;   // Value for output instruction error, ModuleStates local modules
   END_VAR
BEGIN
   //=============================================================================
   //SIEMENS AG
   //(c)Copyright 2015 All Rights Reserved
   //-----------------------------------------------------------------------------
   //Library: -
   //Tested with: S7-1516-3 PN/DP FW 1.7
   //Engineering: TIA Portal V13 SP1
   //Restrictions: -
   //Requirements: -
   //Functionality: Determine hardware identifier and module states from local
   //               modules
   //-----------------------------------------------------------------------------
   //Change log table:
   //Version  Date       Expert in charge Changes applied
   //01.00.00 24.03.2015 Siemens Industry Online Support First released version
   //=============================================================================

   //=============================================================================
   // Determine hardware identifier from LOCAL MODULES
   //=============================================================================
   #statGeoAddr.HWTYPE := #MODULE_OF_PLC;      // Hardware type 4: module
   #statGeoAddr.AREA := #CPU;                  // Area ID 0: CPU
   #statGeoAddr.IOSYSTEM := #CENTRAL_SYSTEM;   // PROFINET IO system
                                               // (0 = central unit in the rack)
   #statGeoAddr.STATION := #CENTRAL_STATION;   // Number of the rack
                                               // if area identifier
                                               //  AREA = 0 (central module).

   FOR #tempModuleNum := 1 TO "MAX_MODULES_LOCAL" DO
     // Slot number
     #statGeoAddr.SLOT := INT_TO_UINT(#tempModuleNum);
     // read LADDR from local modules
     #tempRetValGeo := GEO2LOG(GEOADDR := #statGeoAddr,
                               LADDR => #statGeoLaddr);
     // check Retval
     IF (#tempRetValGeo = 0)
     THEN
       // store LADDR from local modules in diagnostic data block
       #plc.slot[#tempModuleNum].slotLaddr := #statGeoLaddr;
       #statActualCentralModules := #statActualCentralModules + 1;
     ELSE
       // If the return value ist not = 0 --> the device/system/module is not
       // configured --> No error handling
       // set LADDR from local modules to 0 in diagnostic data block
       #plc.slot[#tempModuleNum].slotLaddr := 0;
     END_IF;
     // Store the actual configured devices in the diagnostics DB
     #plc.actualConfiguredCentralModules := #statActualCentralModules;
   END_FOR;


   //=============================================================================
   // Check module states from LOCAL MODULES
   //=============================================================================
   // Check if central module are available - at least one module is always
   // configured, the PLC itself
   IF (#plc.actualConfiguredCentralModules > 1)
   THEN
     // Check the status of the local modules
     #tempRetValModuleStates := ModuleStates(LADDR := #HW_ID_PLC_MODULES,
                                             MODE := #STATE_PROBLEM,
                                             STATE := #statPlcModuleStates);

     // Check if the block call was successful
     IF (#tempRetValModuleStates <> 0)
     THEN
       // Error handling
       #status := #tempRetValModuleStates;
       #instructionError := #ERR_MOD_STAT_CENTRAL;
     ELSE
       ; // Everything is ok!
     END_IF;
   ELSE
     ; // There are no central module configured
   END_IF;

   // The error LED of the PLC is flashing --> Set error state of the PLC
   #plc.errorState := TRUE;


   //=============================================================================
   // set module states from LOCAL MODULES
   //=============================================================================

   // If the first bit in the array is true, at least one module is faulty
   IF (#statPlcModuleStates[0] = TRUE)
   THEN
     // Check which of the modules are faulty
     // PLC modules array starts at index 2 for the first local module
     FOR #tempModuleNum := 2 TO #plc.actualConfiguredCentralModules + 1 DO
       IF (#statPlcModuleStates[#tempModuleNum] = TRUE)
       THEN
         #plc.slot[#tempModuleNum - 1].slotErrorState := TRUE;
       ELSE
         #plc.slot[#tempModuleNum - 1].slotErrorState := FALSE;
       END_IF;
     END_FOR;

   ELSE
     // Everything is ok!
     FOR #tempModuleNum := 1 TO #plc.actualConfiguredCentralModules DO
       #plc.slot[#tempModuleNum].slotErrorState := FALSE;
     END_FOR;

   END_IF;
END_FUNCTION_BLOCK

FUNCTION "CopyToHmiDB" : Void   // FC2081, SCL
{ S7_Optimized_Access := 'TRUE' }
VERSION : 0.1
   VAR_INPUT
      deviceIndex : Int;   // Index for Device
   END_VAR
   VAR_IN_OUT
      plc : "typePlc";   // The diagnostics structure for one PLC
      showPlc : "typeShowPlc";   // The show diagnostics structure for one PLC
      ioSystem : "typeIoSystem";   // The diagnostics structure for one IO System
      showIoSystem : "typeShowIoSystem";   // The show diagnostics structure for one IO System
   END_VAR
   VAR_TEMP
      tempSlotIndex : Int;   // Index for Slot
   END_VAR
   // Ret_Val : return value function
BEGIN
   //=============================================================================
   //SIEMENS AG
   //(c)Copyright 2015 All Rights Reserved
   //-----------------------------------------------------------------------------
   //Library: -
   //Tested with: S7-1516-3 PN/DP FW 1.7
   //Engineering: TIA Portal V13 SP1
   //Restrictions: -
   //Requirements: -
   //Functionality: copy error states from DiagnosticData DB to ShowDiag DB 
   //-----------------------------------------------------------------------------
   //Change log table:
   //Version  Date       Expert in charge Changes applied
   //01.00.00 24.03.2015 Siemens Industry Online Support First released version
   //=============================================================================

   //=============================================================================
   // copy errorstates for PLC
   //=============================================================================
   IF (#deviceIndex = 0)
   THEN
     #showPlc.errorState := #plc.errorState;
     FOR #tempSlotIndex := 1 TO "MAX_MODULES_LOCAL" DO
       #showPlc.slot[#tempSlotIndex].slotErrorState := #plc.slot[#tempSlotIndex].slotErrorState;
     END_FOR;

   //=============================================================================
   // copy errorstates for Devices
   //=============================================================================
   ELSIF (#deviceIndex > 0)
   THEN
     #showIoSystem.device[#deviceIndex].errorState := #ioSystem.device[#deviceIndex].errorState;
     FOR #tempSlotIndex := 0 TO #ioSystem.device[#deviceIndex].actualConfiguredModules DO
       #showIoSystem.device[#deviceIndex].slot[#tempSlotIndex].slotErrorState := #ioSystem.device[#deviceIndex].slot[#tempSlotIndex].slotErrorState;
     END_FOR;

   ELSE
     ;
   END_IF;
END_FUNCTION

FUNCTION "DiagnosticError" : Void   // FC2082, SCL
{ S7_Optimized_Access := 'TRUE' }
VERSION : 0.1
   VAR_INPUT
      ioState : Word;   // IO state of the HW object
      laddr : Hw_Any;   // Hardware identifier
      channel : UInt;   // Channel number
      multiError : Bool;   // =true if more than one error is present
   END_VAR
   VAR_IN_OUT
      plc : "typePlc";   // The diagnostics structure for one PLC
      showPlc : "typeShowPlc";   // The show diagnostics structure for one PLC
      ioSystem : Array[1.."MAX_SYSTEM"] of "typeIoSystem";   // The diagnostics structure for one IO System
      showIoSystem : Array[1.."MAX_SYSTEM"] of "typeShowIoSystem";   // The show diagnostics structure for one IO System
      showActIoSystem : "typeShowActIoSystem";   // The show diagnostics structure for the selected IO System
   END_VAR
   VAR_TEMP
      index : Int;   // index system
      tempIoSystemIndex : Int;   // Index for IO System
      tempGeoAddr : GEOADDR;   // Geographical address of the disturbed Module / Device
      tempRetVal : Int;   // Return value of LOG2GEO
   END_VAR
   // Ret_Val : return value function
   VAR CONSTANT
      GOOD : Word := 16#01;   // Status of the hardware object: Bit 0: Good
      AREA_CENTRAL : UInt := 0;   // Area ID for PLC
      AREA_PROFINET : UInt := 1;   // Area ID for PROFINET IO
      AREA_PROFIBUS : UInt := 2;   // Area ID for PROFIBUS DP
   END_VAR
BEGIN
   //=============================================================================
   //SIEMENS AG
   //(c)Copyright 2015 All Rights Reserved
   //-----------------------------------------------------------------------------
   //Library: -
   //Tested with: S7-1516-3 PN/DP FW 1.7
   //Engineering: TIA Portal V13 SP1
   //Restrictions: -
   //Requirements: -
   //Functionality: Evaluate Diagnostic interrupt OB information for PLC and
   //               devices
   //-----------------------------------------------------------------------------
   //Change log table:
   //Version  Date       Expert in charge Changes applied
   //01.00.00 24.03.2015 Siemens Industry Online Support First released version
   //=============================================================================

   //=============================================================================
   // evaluate IO state from Diagnostic interrupt OB
   // and set information to DiagnosticsData DB
   //=============================================================================

